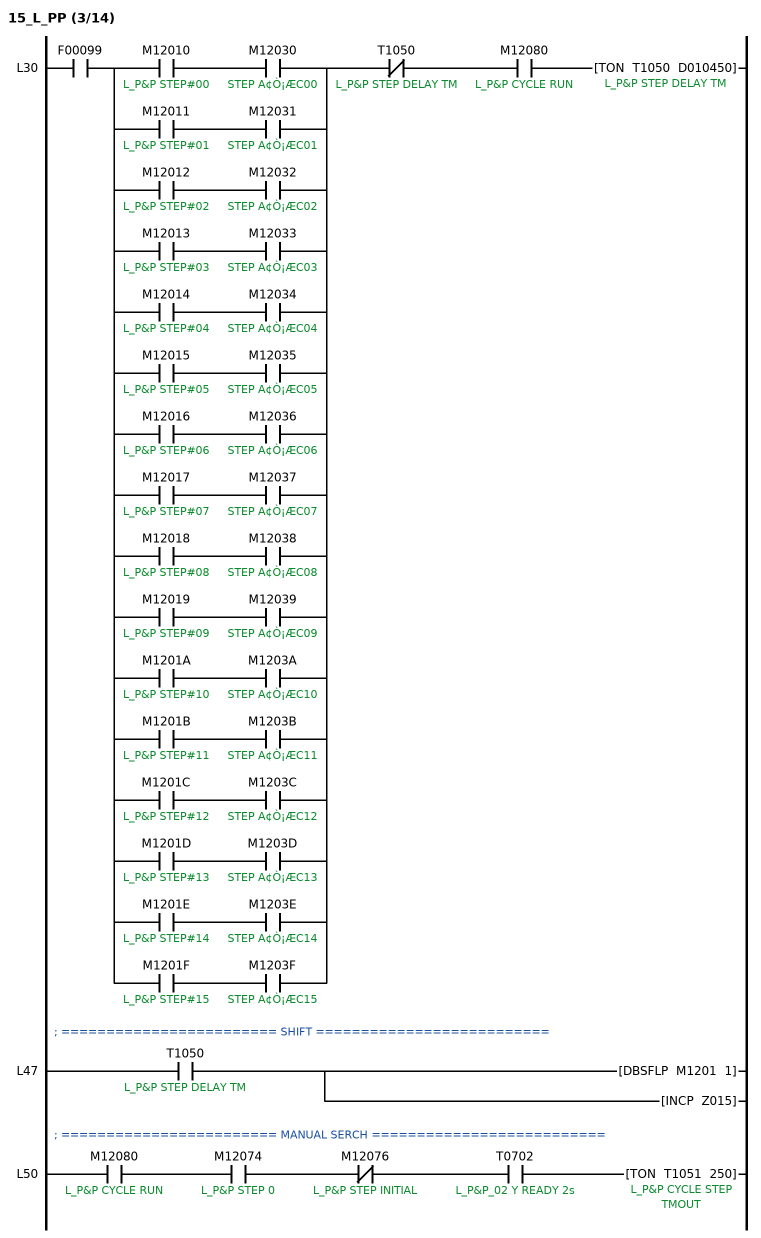
[picture p120: 15_L_PP rungs L30-L50]
; L30
LOAD      F00099
LOAD      M12010	// L_P&P STEP#00
AND       M12030	// STEP A¢Ò¡ÆC00
LOAD      M12011	// L_P&P STEP#01
AND       M12031	// STEP A¢Ò¡ÆC01
OR LOAD
LOAD      M12012	// L_P&P STEP#02
AND       M12032	// STEP A¢Ò¡ÆC02
OR LOAD
LOAD      M12013	// L_P&P STEP#03
AND       M12033	// STEP A¢Ò¡ÆC03
OR LOAD
LOAD      M12014	// L_P&P STEP#04
AND       M12034	// STEP A¢Ò¡ÆC04
OR LOAD
LOAD      M12015	// L_P&P STEP#05
AND       M12035	// STEP A¢Ò¡ÆC05
OR LOAD
LOAD      M12016	// L_P&P STEP#06
AND       M12036	// STEP A¢Ò¡ÆC06
OR LOAD
LOAD      M12017	// L_P&P STEP#07
AND       M12037	// STEP A¢Ò¡ÆC07
OR LOAD
LOAD      M12018	// L_P&P STEP#08
AND       M12038	// STEP A¢Ò¡ÆC08
OR LOAD
LOAD      M12019	// L_P&P STEP#09
AND       M12039	// STEP A¢Ò¡ÆC09
OR LOAD
LOAD      M1201A	// L_P&P STEP#10
AND       M1203A	// STEP A¢Ò¡ÆC10
OR LOAD
LOAD      M1201B	// L_P&P STEP#11
AND       M1203B	// STEP A¢Ò¡ÆC11
OR LOAD
LOAD      M1201C	// L_P&P STEP#12
AND       M1203C	// STEP A¢Ò¡ÆC12
OR LOAD
LOAD      M1201D	// L_P&P STEP#13
AND       M1203D	// STEP A¢Ò¡ÆC13
OR LOAD
LOAD      M1201E	// L_P&P STEP#14
AND       M1203E	// STEP A¢Ò¡ÆC14
OR LOAD
LOAD      M1201F	// L_P&P STEP#15
AND       M1203F	// STEP A¢Ò¡ÆC15
OR LOAD
AND LOAD
AND NOT   T1050	// L_P&P STEP DELAY TM
AND       M12080	// L_P&P CYCLE RUN
TON       T1050 D010450	// L_P&P STEP DELAY TM
// ======================== SHIFT ==========================
; L47
LOAD      T1050	// L_P&P STEP DELAY TM
DBSFLP    M1201 1
INCP      Z015
// ======================== MANUAL SERCH ==========================
; L50
LOAD      M12080	// L_P&P CYCLE RUN
AND       M12074	// L_P&P STEP 0
AND NOT   M12076	// L_P&P STEP INITIAL
AND       T0702	// L_P&P_02 Y READY 2s
TON       T1051 250	// L_P&P CYCLE STEP TMOUT

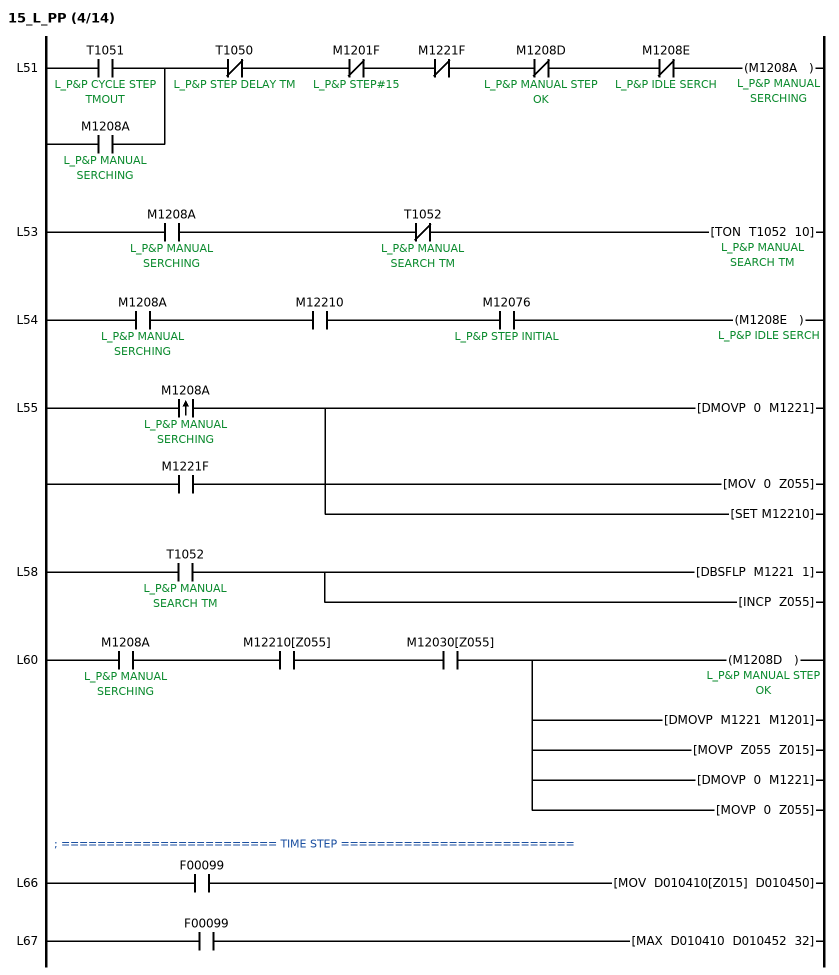
; L51
LOAD      T1051	// L_P&P CYCLE STEP TMOUT
OR        M1208A	// L_P&P MANUAL SERCHING
AND NOT   T1050	// L_P&P STEP DELAY TM
AND NOT   M1201F	// L_P&P STEP#15
AND NOT   M1221F
AND NOT   M1208D	// L_P&P MANUAL STEP OK
AND NOT   M1208E	// L_P&P IDLE SERCH
OUT       M1208A	// L_P&P MANUAL SERCHING
; L53
LOAD      M1208A	// L_P&P MANUAL SERCHING
AND NOT   T1052	// L_P&P MANUAL SEARCH TM
TON       T1052 10	// L_P&P MANUAL SEARCH TM
; L54
LOAD      M1208A	// L_P&P MANUAL SERCHING
AND       M12210
AND       M12076	// L_P&P STEP INITIAL
OUT       M1208E	// L_P&P IDLE SERCH
; L55
LOADP     M1208A	// L_P&P MANUAL SERCHING
OR        M1221F
DMOVP     0 M1221
MOV       0 Z055
SET       M12210
; L58
LOAD      T1052	// L_P&P MANUAL SEARCH TM
DBSFLP    M1221 1
INCP      Z055
; L60
LOAD      M1208A	// L_P&P MANUAL SERCHING
AND       M12210[Z055]
AND       M12030[Z055]
OUT       M1208D	// L_P&P MANUAL STEP OK
DMOVP     M1221 M1201
MOVP      Z055 Z015
DMOVP     0 M1221
MOVP      0 Z055
// ======================== TIME STEP ==========================
; L66
LOAD      F00099
MOV       D010410[Z015] D010450
; L67
LOAD      F00099
MAX       D010410 D010452 32

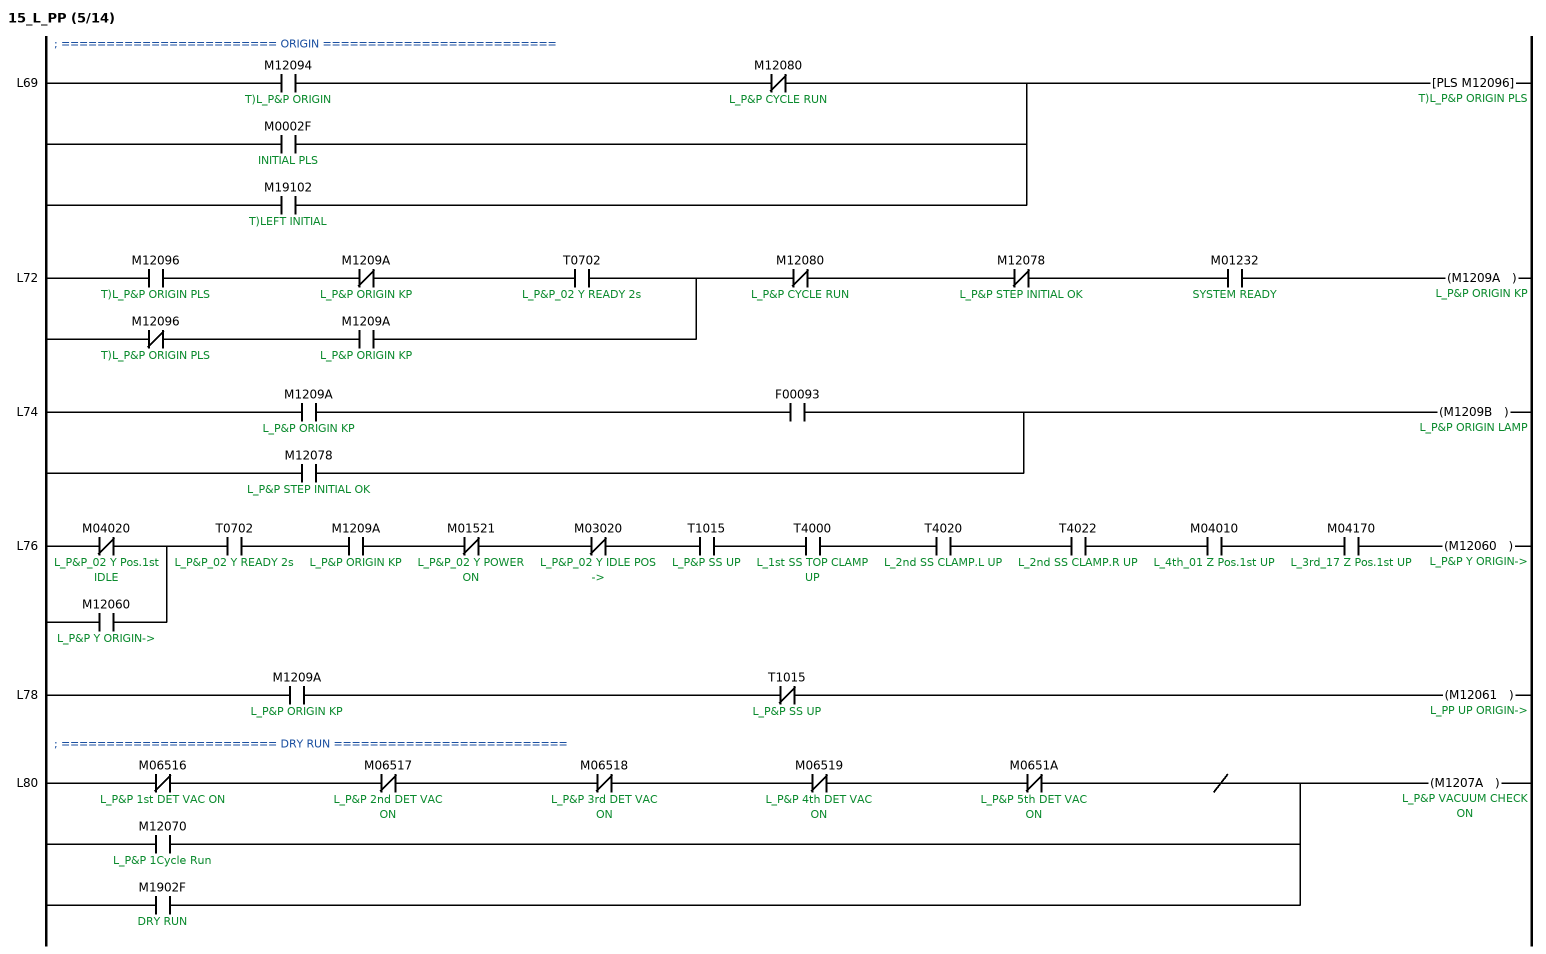
// ======================== ORIGIN ==========================
; L69
LOAD      M12094	// T)L_P&P ORIGIN
AND NOT   M12080	// L_P&P CYCLE RUN
OR        M0002F	// INITIAL PLS
OR        M19102	// T)LEFT INITIAL
OUTP      M12096	// T)L_P&P ORIGIN PLS
; L72
LOAD      M12096	// T)L_P&P ORIGIN PLS
AND NOT   M1209A	// L_P&P ORIGIN KP
AND       T0702	// L_P&P_02 Y READY 2s
LOAD NOT  M12096	// T)L_P&P ORIGIN PLS
AND       M1209A	// L_P&P ORIGIN KP
OR LOAD
AND NOT   M12080	// L_P&P CYCLE RUN
AND NOT   M12078	// L_P&P STEP INITIAL OK
AND       M01232	// SYSTEM READY
OUT       M1209A	// L_P&P ORIGIN KP
; L74
LOAD      M1209A	// L_P&P ORIGIN KP
AND       F00093
OR        M12078	// L_P&P STEP INITIAL OK
OUT       M1209B	// L_P&P ORIGIN LAMP
; L76
LOAD NOT  M04020	// L_P&P_02 Y Pos.1st IDLE
OR        M12060	// L_P&P Y ORIGIN->
AND       T0702	// L_P&P_02 Y READY 2s
AND       M1209A	// L_P&P ORIGIN KP
AND NOT   M01521	// L_P&P_02 Y POWER ON
AND NOT   M03020	// L_P&P_02 Y IDLE POS ->
AND       T1015	// L_P&P SS UP
AND       T4000	// L_1st SS TOP CLAMP    UP
AND       T4020	// L_2nd SS CLAMP.L UP
AND       T4022	// L_2nd SS CLAMP.R UP
AND       M04010	// L_4th_01 Z Pos.1st UP
AND       M04170	// L_3rd_17 Z Pos.1st UP
OUT       M12060	// L_P&P Y ORIGIN->
; L78
LOAD      M1209A	// L_P&P ORIGIN KP
AND NOT   T1015	// L_P&P SS UP
OUT       M12061	// L_PP UP ORIGIN->
// ======================== DRY RUN ==========================
; L80
LOAD NOT  M06516	// L_P&P 1st DET VAC ON
AND NOT   M06517	// L_P&P 2nd DET VAC ON
AND NOT   M06518	// L_P&P 3rd DET VAC ON
AND NOT   M06519	// L_P&P 4th DET VAC ON
AND NOT   M0651A	// L_P&P 5th DET VAC ON
NOT
OR        M12070	// L_P&P 1Cycle Run
OR        M1902F	// DRY RUN
OUT       M1207A	// L_P&P VACUUM CHECK ON

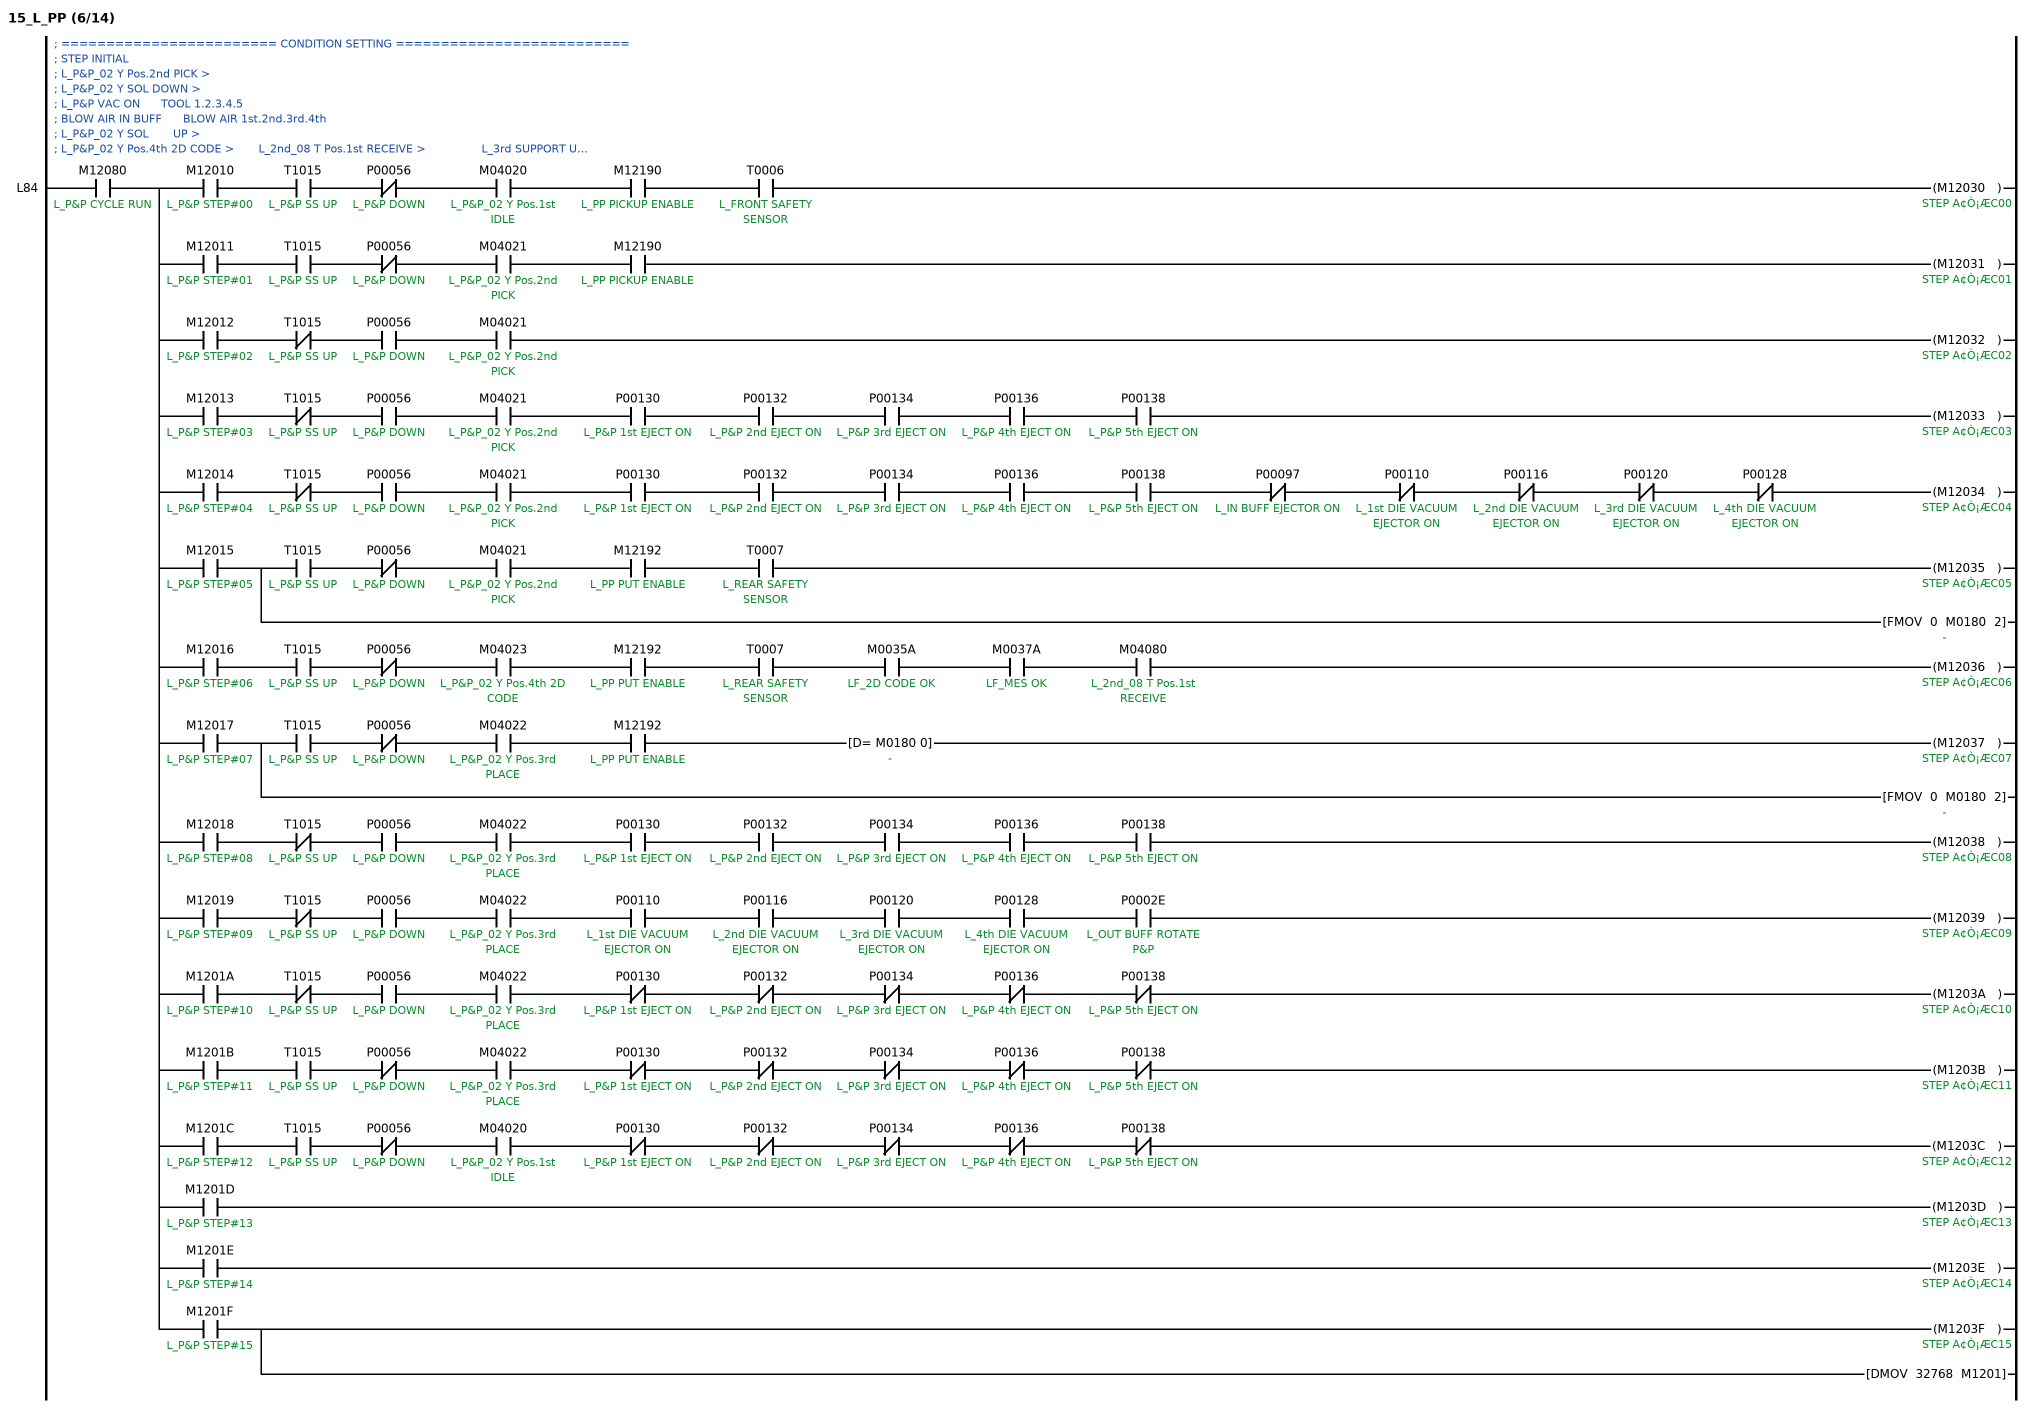
// ======================== CONDITION SETTING ==========================
; L84
LOAD      M12080	// L_P&P CYCLE RUN
MPUSH
AND       M12010	// L_P&P STEP#00
AND       T1015	// L_P&P SS UP
AND NOT   P00056	// L_P&P DOWN
AND       M04020	// L_P&P_02 Y Pos.1st IDLE
AND       M12190	// L_PP PICKUP ENABLE
AND       T0006	// L_FRONT SAFETY SENSOR
OUT       M12030	// STEP A¢Ò¡ÆC00
MLOAD
AND       M12011	// L_P&P STEP#01
AND       T1015	// L_P&P SS UP
AND NOT   P00056	// L_P&P DOWN
AND       M04021	// L_P&P_02 Y Pos.2nd PICK
AND       M12190	// L_PP PICKUP ENABLE
OUT       M12031	// STEP A¢Ò¡ÆC01
MLOAD
AND       M12012	// L_P&P STEP#02
AND NOT   T1015	// L_P&P SS UP
AND       P00056	// L_P&P DOWN
AND       M04021	// L_P&P_02 Y Pos.2nd PICK
OUT       M12032	// STEP A¢Ò¡ÆC02
MLOAD
AND       M12013	// L_P&P STEP#03
AND NOT   T1015	// L_P&P SS UP
AND       P00056	// L_P&P DOWN
AND       M04021	// L_P&P_02 Y Pos.2nd PICK
AND       P00130	// L_P&P 1st EJECT ON
AND       P00132	// L_P&P 2nd EJECT ON
AND       P00134	// L_P&P 3rd EJECT ON
AND       P00136	// L_P&P 4th EJECT ON
AND       P00138	// L_P&P 5th EJECT ON
OUT       M12033	// STEP A¢Ò¡ÆC03
MLOAD
AND       M12014	// L_P&P STEP#04
AND NOT   T1015	// L_P&P SS UP
AND       P00056	// L_P&P DOWN
AND       M04021	// L_P&P_02 Y Pos.2nd PICK
AND       P00130	// L_P&P 1st EJECT ON
AND       P00132	// L_P&P 2nd EJECT ON
AND       P00134	// L_P&P 3rd EJECT ON
AND       P00136	// L_P&P 4th EJECT ON
AND       P00138	// L_P&P 5th EJECT ON
AND NOT   P00097	// L_IN BUFF EJECTOR ON
AND NOT   P00110	// L_1st DIE VACUUM EJECTOR ON
AND NOT   P00116	// L_2nd DIE VACUUM EJECTOR ON
AND NOT   P00120	// L_3rd DIE VACUUM EJECTOR ON
AND NOT   P00128	// L_4th DIE VACUUM EJECTOR ON
OUT       M12034	// STEP A¢Ò¡ÆC04
MLOAD
AND       M12015	// L_P&P STEP#05
MPUSH
AND       T1015	// L_P&P SS UP
AND NOT   P00056	// L_P&P DOWN
AND       M04021	// L_P&P_02 Y Pos.2nd PICK
AND       M12192	// L_PP PUT ENABLE
AND       T0007	// L_REAR SAFETY SENSOR
OUT       M12035	// STEP A¢Ò¡ÆC05
MPOP
FMOV      0 M0180 2	// -
MLOAD
AND       M12016	// L_P&P STEP#06
AND       T1015	// L_P&P SS UP
AND NOT   P00056	// L_P&P DOWN
AND       M04023	// L_P&P_02 Y Pos.4th 2D CODE
AND       M12192	// L_PP PUT ENABLE
AND       T0007	// L_REAR SAFETY SENSOR
AND       M0035A	// LF_2D CODE OK
AND       M0037A	// LF_MES OK
AND       M04080	// L_2nd_08 T Pos.1st RECEIVE
OUT       M12036	// STEP A¢Ò¡ÆC06
MLOAD
AND       M12017	// L_P&P STEP#07
MPUSH
AND       T1015	// L_P&P SS UP
AND NOT   P00056	// L_P&P DOWN
AND       M04022	// L_P&P_02 Y Pos.3rd PLACE
AND       M12192	// L_PP PUT ENABLE
ANDD=     M0180 0	// -
OUT       M12037	// STEP A¢Ò¡ÆC07
MPOP
FMOV      0 M0180 2	// -
MLOAD
AND       M12018	// L_P&P STEP#08
AND NOT   T1015	// L_P&P SS UP
AND       P00056	// L_P&P DOWN
AND       M04022	// L_P&P_02 Y Pos.3rd PLACE
AND       P00130	// L_P&P 1st EJECT ON
AND       P00132	// L_P&P 2nd EJECT ON
AND       P00134	// L_P&P 3rd EJECT ON
AND       P00136	// L_P&P 4th EJECT ON
AND       P00138	// L_P&P 5th EJECT ON
OUT       M12038	// STEP A¢Ò¡ÆC08
MLOAD
AND       M12019	// L_P&P STEP#09
AND NOT   T1015	// L_P&P SS UP
AND       P00056	// L_P&P DOWN
AND       M04022	// L_P&P_02 Y Pos.3rd PLACE
AND       P00110	// L_1st DIE VACUUM EJECTOR ON
AND       P00116	// L_2nd DIE VACUUM EJECTOR ON
AND       P00120	// L_3rd DIE VACUUM EJECTOR ON
AND       P00128	// L_4th DIE VACUUM EJECTOR ON
AND       P0002E	// L_OUT BUFF ROTATE      P&P
OUT       M12039	// STEP A¢Ò¡ÆC09
MLOAD
AND       M1201A	// L_P&P STEP#10
AND NOT   T1015	// L_P&P SS UP
AND       P00056	// L_P&P DOWN
AND       M04022	// L_P&P_02 Y Pos.3rd PLACE
AND NOT   P00130	// L_P&P 1st EJECT ON
AND NOT   P00132	// L_P&P 2nd EJECT ON
AND NOT   P00134	// L_P&P 3rd EJECT ON
AND NOT   P00136	// L_P&P 4th EJECT ON
AND NOT   P00138	// L_P&P 5th EJECT ON
OUT       M1203A	// STEP A¢Ò¡ÆC10
MLOAD
AND       M1201B	// L_P&P STEP#11
AND       T1015	// L_P&P SS UP
AND NOT   P00056	// L_P&P DOWN
AND       M04022	// L_P&P_02 Y Pos.3rd PLACE
AND NOT   P00130	// L_P&P 1st EJECT ON
AND NOT   P00132	// L_P&P 2nd EJECT ON
AND NOT   P00134	// L_P&P 3rd EJECT ON
AND NOT   P00136	// L_P&P 4th EJECT ON
AND NOT   P00138	// L_P&P 5th EJECT ON
OUT       M1203B	// STEP A¢Ò¡ÆC11
MLOAD
AND       M1201C	// L_P&P STEP#12
AND       T1015	// L_P&P SS UP
AND NOT   P00056	// L_P&P DOWN
AND       M04020	// L_P&P_02 Y Pos.1st IDLE
AND NOT   P00130	// L_P&P 1st EJECT ON
AND NOT   P00132	// L_P&P 2nd EJECT ON
AND NOT   P00134	// L_P&P 3rd EJECT ON
AND NOT   P00136	// L_P&P 4th EJECT ON
AND NOT   P00138	// L_P&P 5th EJECT ON
OUT       M1203C	// STEP A¢Ò¡ÆC12
MLOAD
AND       M1201D	// L_P&P STEP#13
OUT       M1203D	// STEP A¢Ò¡ÆC13
MLOAD
AND       M1201E	// L_P&P STEP#14
OUT       M1203E	// STEP A¢Ò¡ÆC14
MPOP
AND       M1201F	// L_P&P STEP#15
OUT       M1203F	// STEP A¢Ò¡ÆC15
DMOV      32768 M1201
// output comment: STEP INITIAL
// output comment: L_P&P_02 Y Pos.2nd PICK >
// output comment: L_P&P_02 Y SOL DOWN >
// output comment: L_P&P VAC ON      TOOL 1.2.3.4.5
// output comment: BLOW AIR IN BUFF      BLOW AIR 1st.2nd.3rd.4th
// output comment: L_P&P_02 Y SOL       UP >
// output comment: L_P&P_02 Y Pos.4th 2D CODE >       L_2nd_08 T Pos.1st RECEIVE >                L_3rd SUPPORT UP
// output comment: L_P&P_02 Y Pos.3rd PLACE >
// output comment: L_P&P_02 Y SOL       DOWN >
// output comment: L_P&P BLOW AIR      TOOL 1.2.3.4.5
// output comment: L_P&P_02 Y SOL       UP >
// output comment: L_P&P_02 Y Pos.1st IDLE >

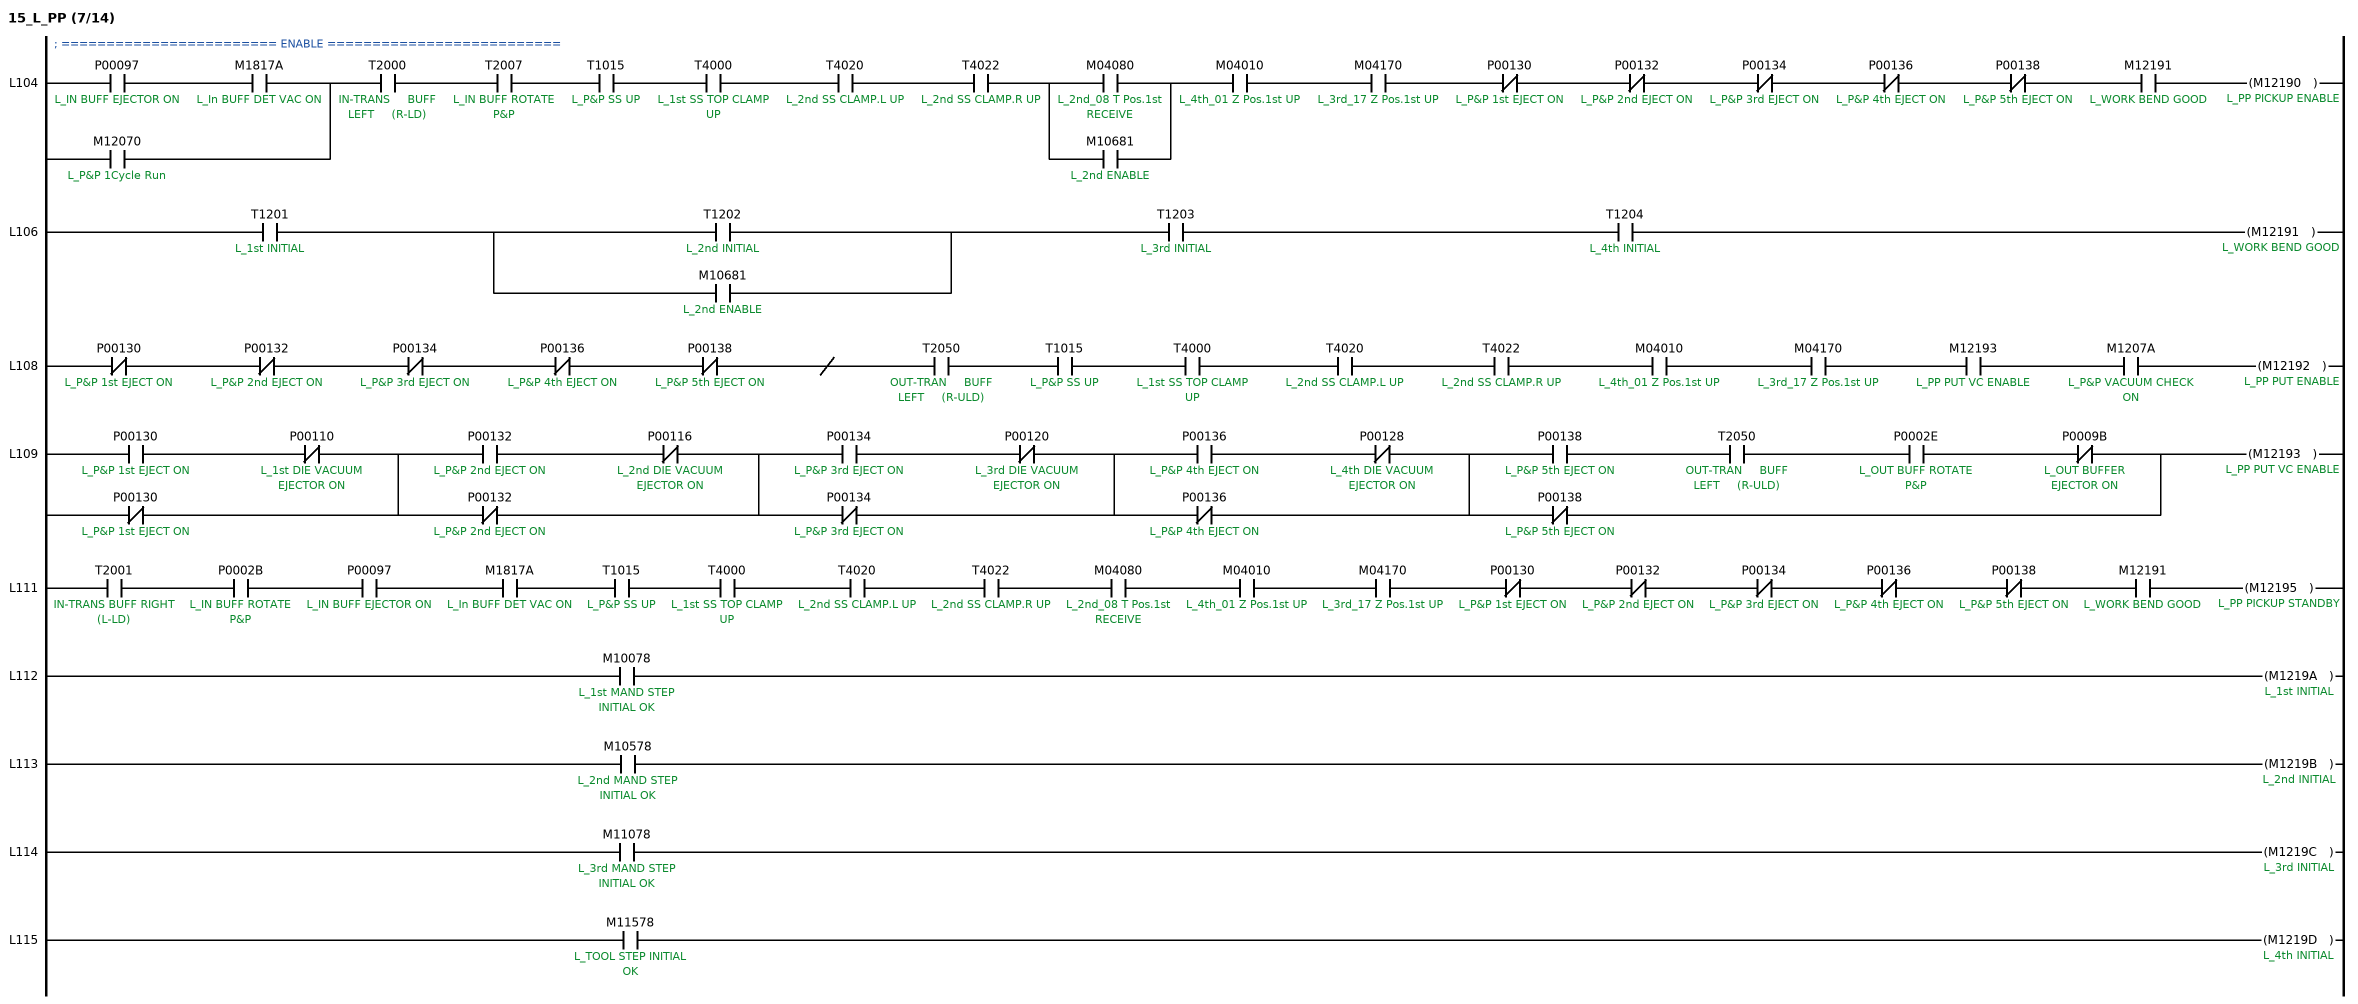
// ======================== ENABLE ==========================
; L104
LOAD      P00097	// L_IN BUFF EJECTOR ON
AND       M1817A	// L_In BUFF DET VAC ON
OR        M12070	// L_P&P 1Cycle Run
AND       T2000	// IN-TRANS     BUFF     LEFT     (R-LD)
AND       T2007	// L_IN BUFF ROTATE      P&P
AND       T1015	// L_P&P SS UP
AND       T4000	// L_1st SS TOP CLAMP    UP
AND       T4020	// L_2nd SS CLAMP.L UP
AND       T4022	// L_2nd SS CLAMP.R UP
LOAD      M04080	// L_2nd_08 T Pos.1st RECEIVE
OR        M10681	// L_2nd ENABLE
AND LOAD
AND       M04010	// L_4th_01 Z Pos.1st UP
AND       M04170	// L_3rd_17 Z Pos.1st UP
AND NOT   P00130	// L_P&P 1st EJECT ON
AND NOT   P00132	// L_P&P 2nd EJECT ON
AND NOT   P00134	// L_P&P 3rd EJECT ON
AND NOT   P00136	// L_P&P 4th EJECT ON
AND NOT   P00138	// L_P&P 5th EJECT ON
AND       M12191	// L_WORK BEND GOOD
OUT       M12190	// L_PP PICKUP ENABLE
; L106
LOAD      T1201	// L_1st INITIAL
LOAD      T1202	// L_2nd INITIAL
OR        M10681	// L_2nd ENABLE
AND LOAD
AND       T1203	// L_3rd INITIAL
AND       T1204	// L_4th INITIAL
OUT       M12191	// L_WORK BEND GOOD
; L108
LOAD NOT  P00130	// L_P&P 1st EJECT ON
AND NOT   P00132	// L_P&P 2nd EJECT ON
AND NOT   P00134	// L_P&P 3rd EJECT ON
AND NOT   P00136	// L_P&P 4th EJECT ON
AND NOT   P00138	// L_P&P 5th EJECT ON
NOT
AND       T2050	// OUT-TRAN     BUFF     LEFT     (R-ULD)
AND       T1015	// L_P&P SS UP
AND       T4000	// L_1st SS TOP CLAMP    UP
AND       T4020	// L_2nd SS CLAMP.L UP
AND       T4022	// L_2nd SS CLAMP.R UP
AND       M04010	// L_4th_01 Z Pos.1st UP
AND       M04170	// L_3rd_17 Z Pos.1st UP
AND       M12193	// L_PP PUT VC ENABLE
AND       M1207A	// L_P&P VACUUM CHECK ON
OUT       M12192	// L_PP PUT ENABLE
; L109
LOAD      P00130	// L_P&P 1st EJECT ON
AND NOT   P00110	// L_1st DIE VACUUM EJECTOR ON
OR NOT    P00130	// L_P&P 1st EJECT ON
LOAD      P00132	// L_P&P 2nd EJECT ON
AND NOT   P00116	// L_2nd DIE VACUUM EJECTOR ON
OR NOT    P00132	// L_P&P 2nd EJECT ON
AND LOAD
LOAD      P00134	// L_P&P 3rd EJECT ON
AND NOT   P00120	// L_3rd DIE VACUUM EJECTOR ON
OR NOT    P00134	// L_P&P 3rd EJECT ON
AND LOAD
LOAD      P00136	// L_P&P 4th EJECT ON
AND NOT   P00128	// L_4th DIE VACUUM EJECTOR ON
OR NOT    P00136	// L_P&P 4th EJECT ON
AND LOAD
LOAD      P00138	// L_P&P 5th EJECT ON
AND       T2050	// OUT-TRAN     BUFF     LEFT     (R-ULD)
AND       P0002E	// L_OUT BUFF ROTATE      P&P
AND NOT   P0009B	// L_OUT BUFFER EJECTOR ON
OR NOT    P00138	// L_P&P 5th EJECT ON
AND LOAD
OUT       M12193	// L_PP PUT VC ENABLE
; L111
LOAD      T2001	// IN-TRANS BUFF RIGHT     (L-LD)
AND       P0002B	// L_IN BUFF ROTATE      P&P
AND       P00097	// L_IN BUFF EJECTOR ON
AND       M1817A	// L_In BUFF DET VAC ON
AND       T1015	// L_P&P SS UP
AND       T4000	// L_1st SS TOP CLAMP    UP
AND       T4020	// L_2nd SS CLAMP.L UP
AND       T4022	// L_2nd SS CLAMP.R UP
AND       M04080	// L_2nd_08 T Pos.1st RECEIVE
AND       M04010	// L_4th_01 Z Pos.1st UP
AND       M04170	// L_3rd_17 Z Pos.1st UP
AND NOT   P00130	// L_P&P 1st EJECT ON
AND NOT   P00132	// L_P&P 2nd EJECT ON
AND NOT   P00134	// L_P&P 3rd EJECT ON
AND NOT   P00136	// L_P&P 4th EJECT ON
AND NOT   P00138	// L_P&P 5th EJECT ON
AND       M12191	// L_WORK BEND GOOD
OUT       M12195	// L_PP PICKUP STANDBY
; L112
LOAD      M10078	// L_1st MAND STEP INITIAL OK
OUT       M1219A	// L_1st INITIAL
; L113
LOAD      M10578	// L_2nd MAND STEP INITIAL OK
OUT       M1219B	// L_2nd INITIAL
; L114
LOAD      M11078	// L_3rd MAND STEP INITIAL OK
OUT       M1219C	// L_3rd INITIAL
; L115
LOAD      M11578	// L_TOOL STEP INITIAL OK
OUT       M1219D	// L_4th INITIAL

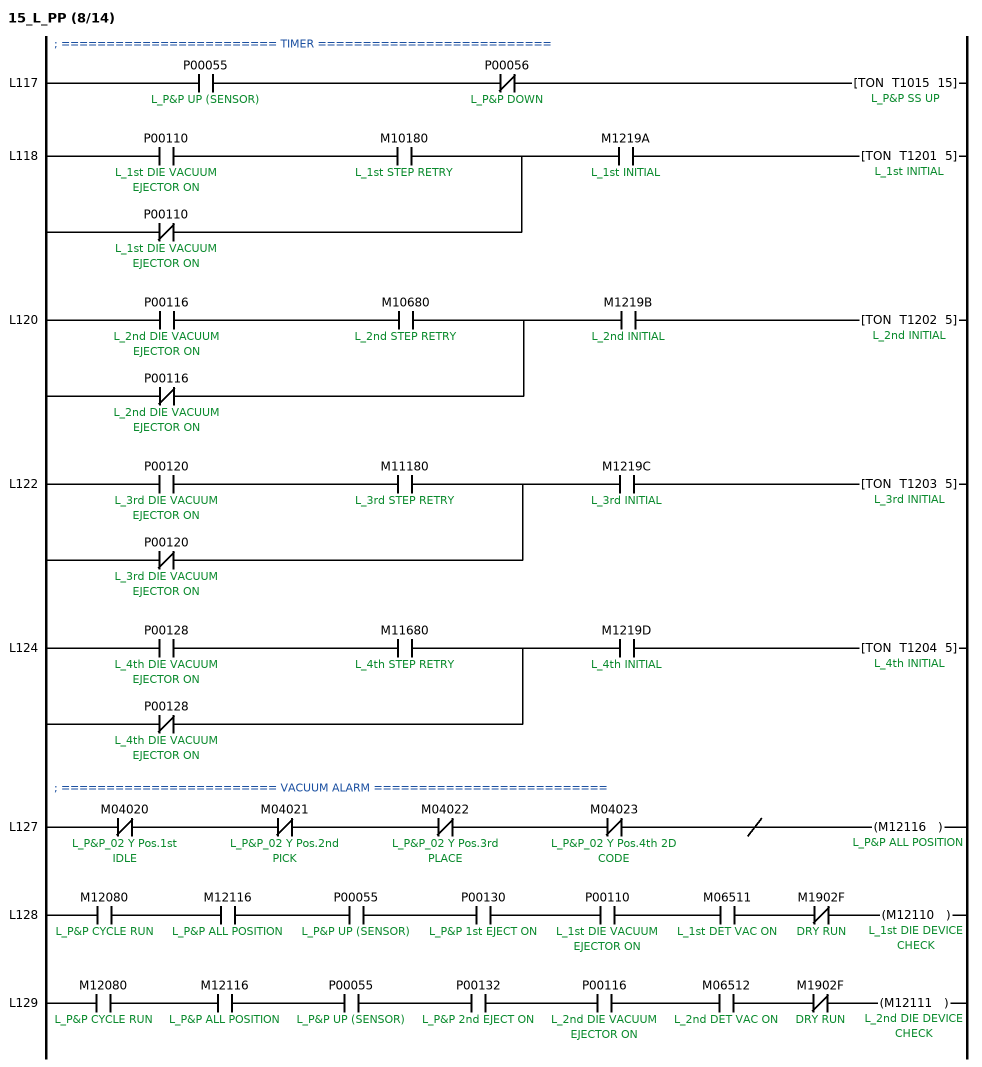
// ======================== TIMER ==========================
; L117
LOAD      P00055	// L_P&P UP (SENSOR)
AND NOT   P00056	// L_P&P DOWN
TON       T1015 15	// L_P&P SS UP
; L118
LOAD      P00110	// L_1st DIE VACUUM EJECTOR ON
AND       M10180	// L_1st STEP RETRY
OR NOT    P00110	// L_1st DIE VACUUM EJECTOR ON
AND       M1219A	// L_1st INITIAL
TON       T1201 5	// L_1st INITIAL
; L120
LOAD      P00116	// L_2nd DIE VACUUM EJECTOR ON
AND       M10680	// L_2nd STEP RETRY
OR NOT    P00116	// L_2nd DIE VACUUM EJECTOR ON
AND       M1219B	// L_2nd INITIAL
TON       T1202 5	// L_2nd INITIAL
; L122
LOAD      P00120	// L_3rd DIE VACUUM EJECTOR ON
AND       M11180	// L_3rd STEP RETRY
OR NOT    P00120	// L_3rd DIE VACUUM EJECTOR ON
AND       M1219C	// L_3rd INITIAL
TON       T1203 5	// L_3rd INITIAL
; L124
LOAD      P00128	// L_4th DIE VACUUM EJECTOR ON
AND       M11680	// L_4th STEP RETRY
OR NOT    P00128	// L_4th DIE VACUUM EJECTOR ON
AND       M1219D	// L_4th INITIAL
TON       T1204 5	// L_4th INITIAL
// ======================== VACUUM ALARM ==========================
; L127
LOAD NOT  M04020	// L_P&P_02 Y Pos.1st IDLE
AND NOT   M04021	// L_P&P_02 Y Pos.2nd PICK
AND NOT   M04022	// L_P&P_02 Y Pos.3rd PLACE
AND NOT   M04023	// L_P&P_02 Y Pos.4th 2D CODE
NOT
OUT       M12116	// L_P&P ALL POSITION
; L128
LOAD      M12080	// L_P&P CYCLE RUN
AND       M12116	// L_P&P ALL POSITION
AND       P00055	// L_P&P UP (SENSOR)
AND       P00130	// L_P&P 1st EJECT ON
AND       P00110	// L_1st DIE VACUUM EJECTOR ON
AND       M06511	// L_1st DET VAC ON
AND NOT   M1902F	// DRY RUN
OUT       M12110	// L_1st DIE DEVICE CHECK
; L129
LOAD      M12080	// L_P&P CYCLE RUN
AND       M12116	// L_P&P ALL POSITION
AND       P00055	// L_P&P UP (SENSOR)
AND       P00132	// L_P&P 2nd EJECT ON
AND       P00116	// L_2nd DIE VACUUM EJECTOR ON
AND       M06512	// L_2nd DET VAC ON
AND NOT   M1902F	// DRY RUN
OUT       M12111	// L_2nd DIE DEVICE CHECK

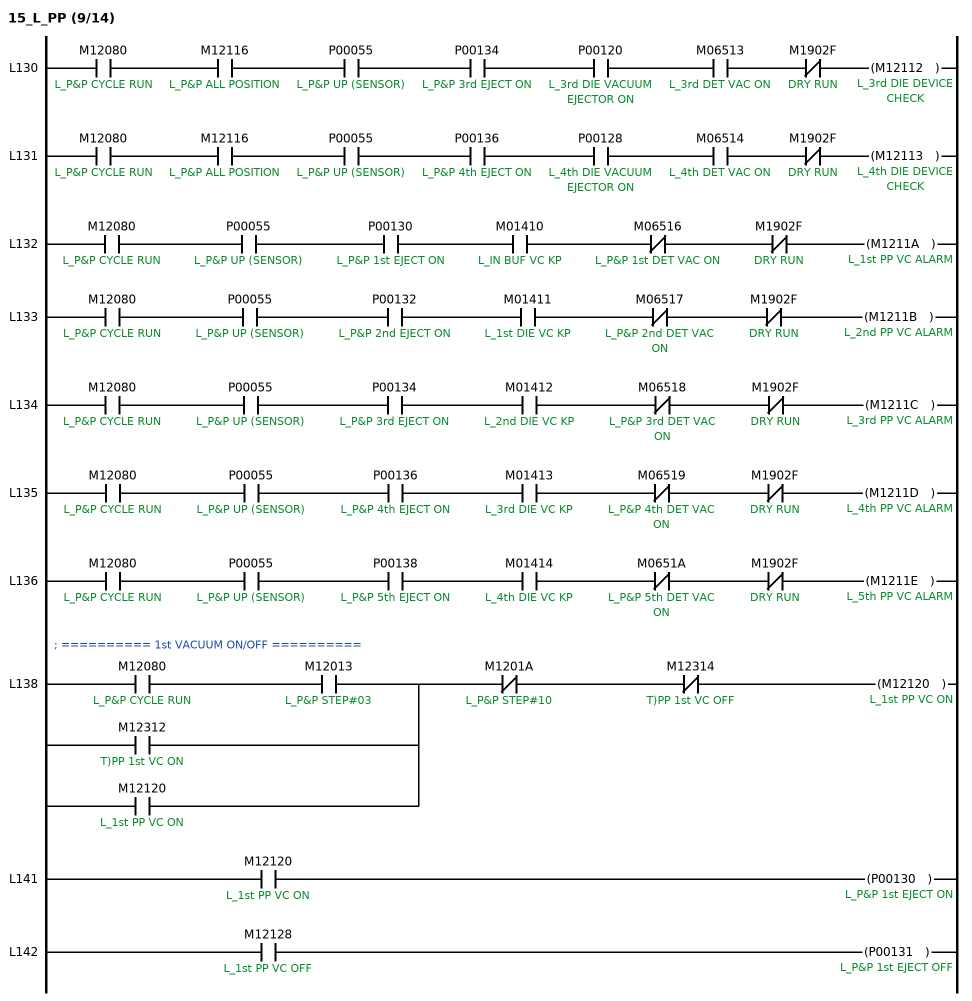
; L130
LOAD      M12080	// L_P&P CYCLE RUN
AND       M12116	// L_P&P ALL POSITION
AND       P00055	// L_P&P UP (SENSOR)
AND       P00134	// L_P&P 3rd EJECT ON
AND       P00120	// L_3rd DIE VACUUM EJECTOR ON
AND       M06513	// L_3rd DET VAC ON
AND NOT   M1902F	// DRY RUN
OUT       M12112	// L_3rd DIE DEVICE CHECK
; L131
LOAD      M12080	// L_P&P CYCLE RUN
AND       M12116	// L_P&P ALL POSITION
AND       P00055	// L_P&P UP (SENSOR)
AND       P00136	// L_P&P 4th EJECT ON
AND       P00128	// L_4th DIE VACUUM EJECTOR ON
AND       M06514	// L_4th DET VAC ON
AND NOT   M1902F	// DRY RUN
OUT       M12113	// L_4th DIE DEVICE CHECK
; L132
LOAD      M12080	// L_P&P CYCLE RUN
AND       P00055	// L_P&P UP (SENSOR)
AND       P00130	// L_P&P 1st EJECT ON
AND       M01410	// L_IN BUF VC KP
AND NOT   M06516	// L_P&P 1st DET VAC ON
AND NOT   M1902F	// DRY RUN
OUT       M1211A	// L_1st PP VC ALARM
; L133
LOAD      M12080	// L_P&P CYCLE RUN
AND       P00055	// L_P&P UP (SENSOR)
AND       P00132	// L_P&P 2nd EJECT ON
AND       M01411	// L_1st DIE VC KP
AND NOT   M06517	// L_P&P 2nd DET VAC ON
AND NOT   M1902F	// DRY RUN
OUT       M1211B	// L_2nd PP VC ALARM
; L134
LOAD      M12080	// L_P&P CYCLE RUN
AND       P00055	// L_P&P UP (SENSOR)
AND       P00134	// L_P&P 3rd EJECT ON
AND       M01412	// L_2nd DIE VC KP
AND NOT   M06518	// L_P&P 3rd DET VAC ON
AND NOT   M1902F	// DRY RUN
OUT       M1211C	// L_3rd PP VC ALARM
; L135
LOAD      M12080	// L_P&P CYCLE RUN
AND       P00055	// L_P&P UP (SENSOR)
AND       P00136	// L_P&P 4th EJECT ON
AND       M01413	// L_3rd DIE VC KP
AND NOT   M06519	// L_P&P 4th DET VAC ON
AND NOT   M1902F	// DRY RUN
OUT       M1211D	// L_4th PP VC ALARM
; L136
LOAD      M12080	// L_P&P CYCLE RUN
AND       P00055	// L_P&P UP (SENSOR)
AND       P00138	// L_P&P 5th EJECT ON
AND       M01414	// L_4th DIE VC KP
AND NOT   M0651A	// L_P&P 5th DET VAC ON
AND NOT   M1902F	// DRY RUN
OUT       M1211E	// L_5th PP VC ALARM
// ========== 1st VACUUM ON/OFF ==========
; L138
LOAD      M12080	// L_P&P CYCLE RUN
AND       M12013	// L_P&P STEP#03
OR        M12312	// T)PP 1st VC ON
OR        M12120	// L_1st PP VC ON
AND NOT   M1201A	// L_P&P STEP#10
AND NOT   M12314	// T)PP 1st VC OFF
OUT       M12120	// L_1st PP VC ON
; L141
LOAD      M12120	// L_1st PP VC ON
OUT       P00130	// L_P&P 1st EJECT ON
; L142
LOAD      M12128	// L_1st PP VC OFF
OUT       P00131	// L_P&P 1st EJECT OFF

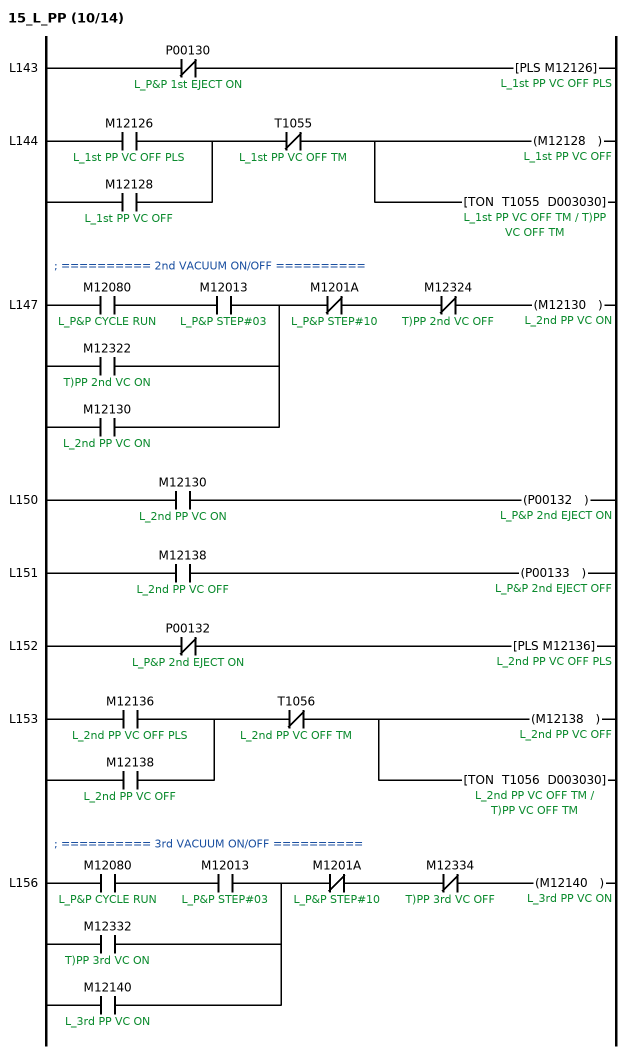
; L143
LOAD NOT  P00130	// L_P&P 1st EJECT ON
OUTP      M12126	// L_1st PP VC OFF PLS
; L144
LOAD      M12126	// L_1st PP VC OFF PLS
OR        M12128	// L_1st PP VC OFF
AND NOT   T1055	// L_1st PP VC OFF TM
OUT       M12128	// L_1st PP VC OFF
TON       T1055 D003030	// L_1st PP VC OFF TM / T)PP VC OFF TM
// ========== 2nd VACUUM ON/OFF ==========
; L147
LOAD      M12080	// L_P&P CYCLE RUN
AND       M12013	// L_P&P STEP#03
OR        M12322	// T)PP 2nd VC ON
OR        M12130	// L_2nd PP VC ON
AND NOT   M1201A	// L_P&P STEP#10
AND NOT   M12324	// T)PP 2nd VC OFF
OUT       M12130	// L_2nd PP VC ON
; L150
LOAD      M12130	// L_2nd PP VC ON
OUT       P00132	// L_P&P 2nd EJECT ON
; L151
LOAD      M12138	// L_2nd PP VC OFF
OUT       P00133	// L_P&P 2nd EJECT OFF
; L152
LOAD NOT  P00132	// L_P&P 2nd EJECT ON
OUTP      M12136	// L_2nd PP VC OFF PLS
; L153
LOAD      M12136	// L_2nd PP VC OFF PLS
OR        M12138	// L_2nd PP VC OFF
AND NOT   T1056	// L_2nd PP VC OFF TM
OUT       M12138	// L_2nd PP VC OFF
TON       T1056 D003030	// L_2nd PP VC OFF TM / T)PP VC OFF TM
// ========== 3rd VACUUM ON/OFF ==========
; L156
LOAD      M12080	// L_P&P CYCLE RUN
AND       M12013	// L_P&P STEP#03
OR        M12332	// T)PP 3rd VC ON
OR        M12140	// L_3rd PP VC ON
AND NOT   M1201A	// L_P&P STEP#10
AND NOT   M12334	// T)PP 3rd VC OFF
OUT       M12140	// L_3rd PP VC ON

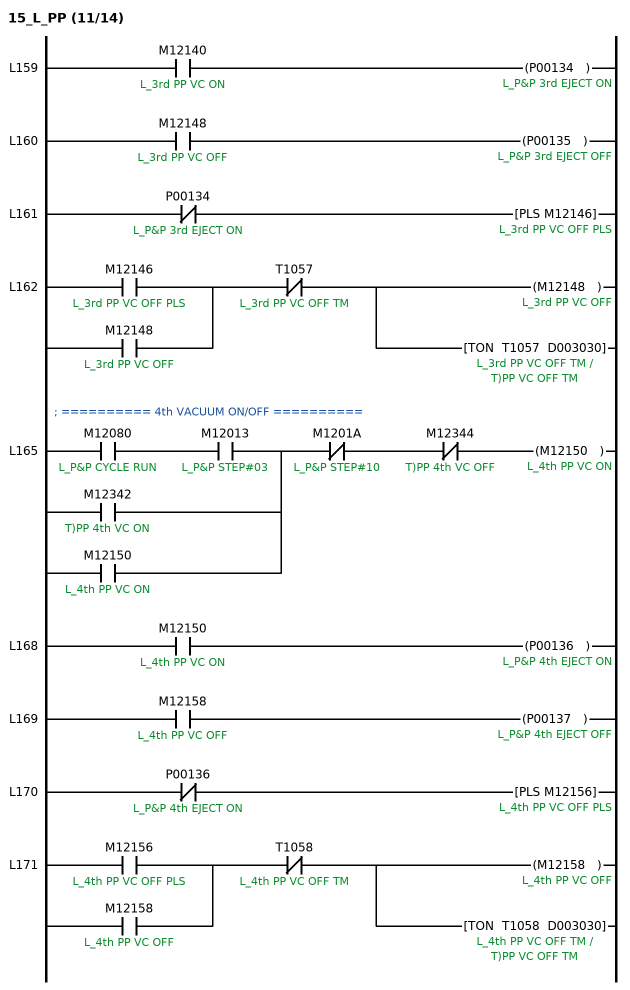
; L159
LOAD      M12140	// L_3rd PP VC ON
OUT       P00134	// L_P&P 3rd EJECT ON
; L160
LOAD      M12148	// L_3rd PP VC OFF
OUT       P00135	// L_P&P 3rd EJECT OFF
; L161
LOAD NOT  P00134	// L_P&P 3rd EJECT ON
OUTP      M12146	// L_3rd PP VC OFF PLS
; L162
LOAD      M12146	// L_3rd PP VC OFF PLS
OR        M12148	// L_3rd PP VC OFF
AND NOT   T1057	// L_3rd PP VC OFF TM
OUT       M12148	// L_3rd PP VC OFF
TON       T1057 D003030	// L_3rd PP VC OFF TM / T)PP VC OFF TM
// ========== 4th VACUUM ON/OFF ==========
; L165
LOAD      M12080	// L_P&P CYCLE RUN
AND       M12013	// L_P&P STEP#03
OR        M12342	// T)PP 4th VC ON
OR        M12150	// L_4th PP VC ON
AND NOT   M1201A	// L_P&P STEP#10
AND NOT   M12344	// T)PP 4th VC OFF
OUT       M12150	// L_4th PP VC ON
; L168
LOAD      M12150	// L_4th PP VC ON
OUT       P00136	// L_P&P 4th EJECT ON
; L169
LOAD      M12158	// L_4th PP VC OFF
OUT       P00137	// L_P&P 4th EJECT OFF
; L170
LOAD NOT  P00136	// L_P&P 4th EJECT ON
OUTP      M12156	// L_4th PP VC OFF PLS
; L171
LOAD      M12156	// L_4th PP VC OFF PLS
OR        M12158	// L_4th PP VC OFF
AND NOT   T1058	// L_4th PP VC OFF TM
OUT       M12158	// L_4th PP VC OFF
TON       T1058 D003030	// L_4th PP VC OFF TM / T)PP VC OFF TM

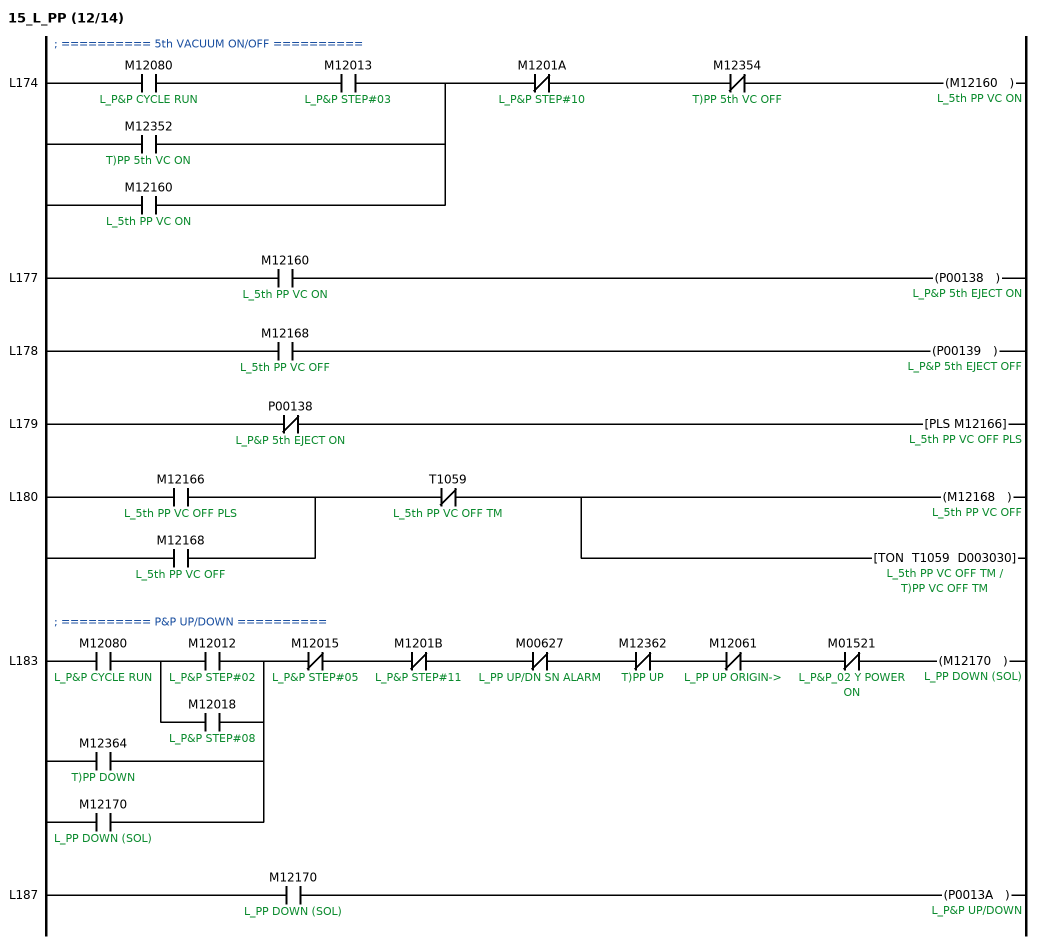
// ========== 5th VACUUM ON/OFF ==========
; L174
LOAD      M12080	// L_P&P CYCLE RUN
AND       M12013	// L_P&P STEP#03
OR        M12352	// T)PP 5th VC ON
OR        M12160	// L_5th PP VC ON
AND NOT   M1201A	// L_P&P STEP#10
AND NOT   M12354	// T)PP 5th VC OFF
OUT       M12160	// L_5th PP VC ON
; L177
LOAD      M12160	// L_5th PP VC ON
OUT       P00138	// L_P&P 5th EJECT ON
; L178
LOAD      M12168	// L_5th PP VC OFF
OUT       P00139	// L_P&P 5th EJECT OFF
; L179
LOAD NOT  P00138	// L_P&P 5th EJECT ON
OUTP      M12166	// L_5th PP VC OFF PLS
; L180
LOAD      M12166	// L_5th PP VC OFF PLS
OR        M12168	// L_5th PP VC OFF
AND NOT   T1059	// L_5th PP VC OFF TM
OUT       M12168	// L_5th PP VC OFF
TON       T1059 D003030	// L_5th PP VC OFF TM / T)PP VC OFF TM
// ========== P&P UP/DOWN ==========
; L183
LOAD      M12080	// L_P&P CYCLE RUN
LOAD      M12012	// L_P&P STEP#02
OR        M12018	// L_P&P STEP#08
AND LOAD
OR        M12364	// T)PP DOWN
OR        M12170	// L_PP DOWN (SOL)
AND NOT   M12015	// L_P&P STEP#05
AND NOT   M1201B	// L_P&P STEP#11
AND NOT   M00627	// L_PP UP/DN SN ALARM
AND NOT   M12362	// T)PP UP
AND NOT   M12061	// L_PP UP ORIGIN->
AND NOT   M01521	// L_P&P_02 Y POWER ON
OUT       M12170	// L_PP DOWN (SOL)
; L187
LOAD      M12170	// L_PP DOWN (SOL)
OUT       P0013A	// L_P&P UP/DOWN

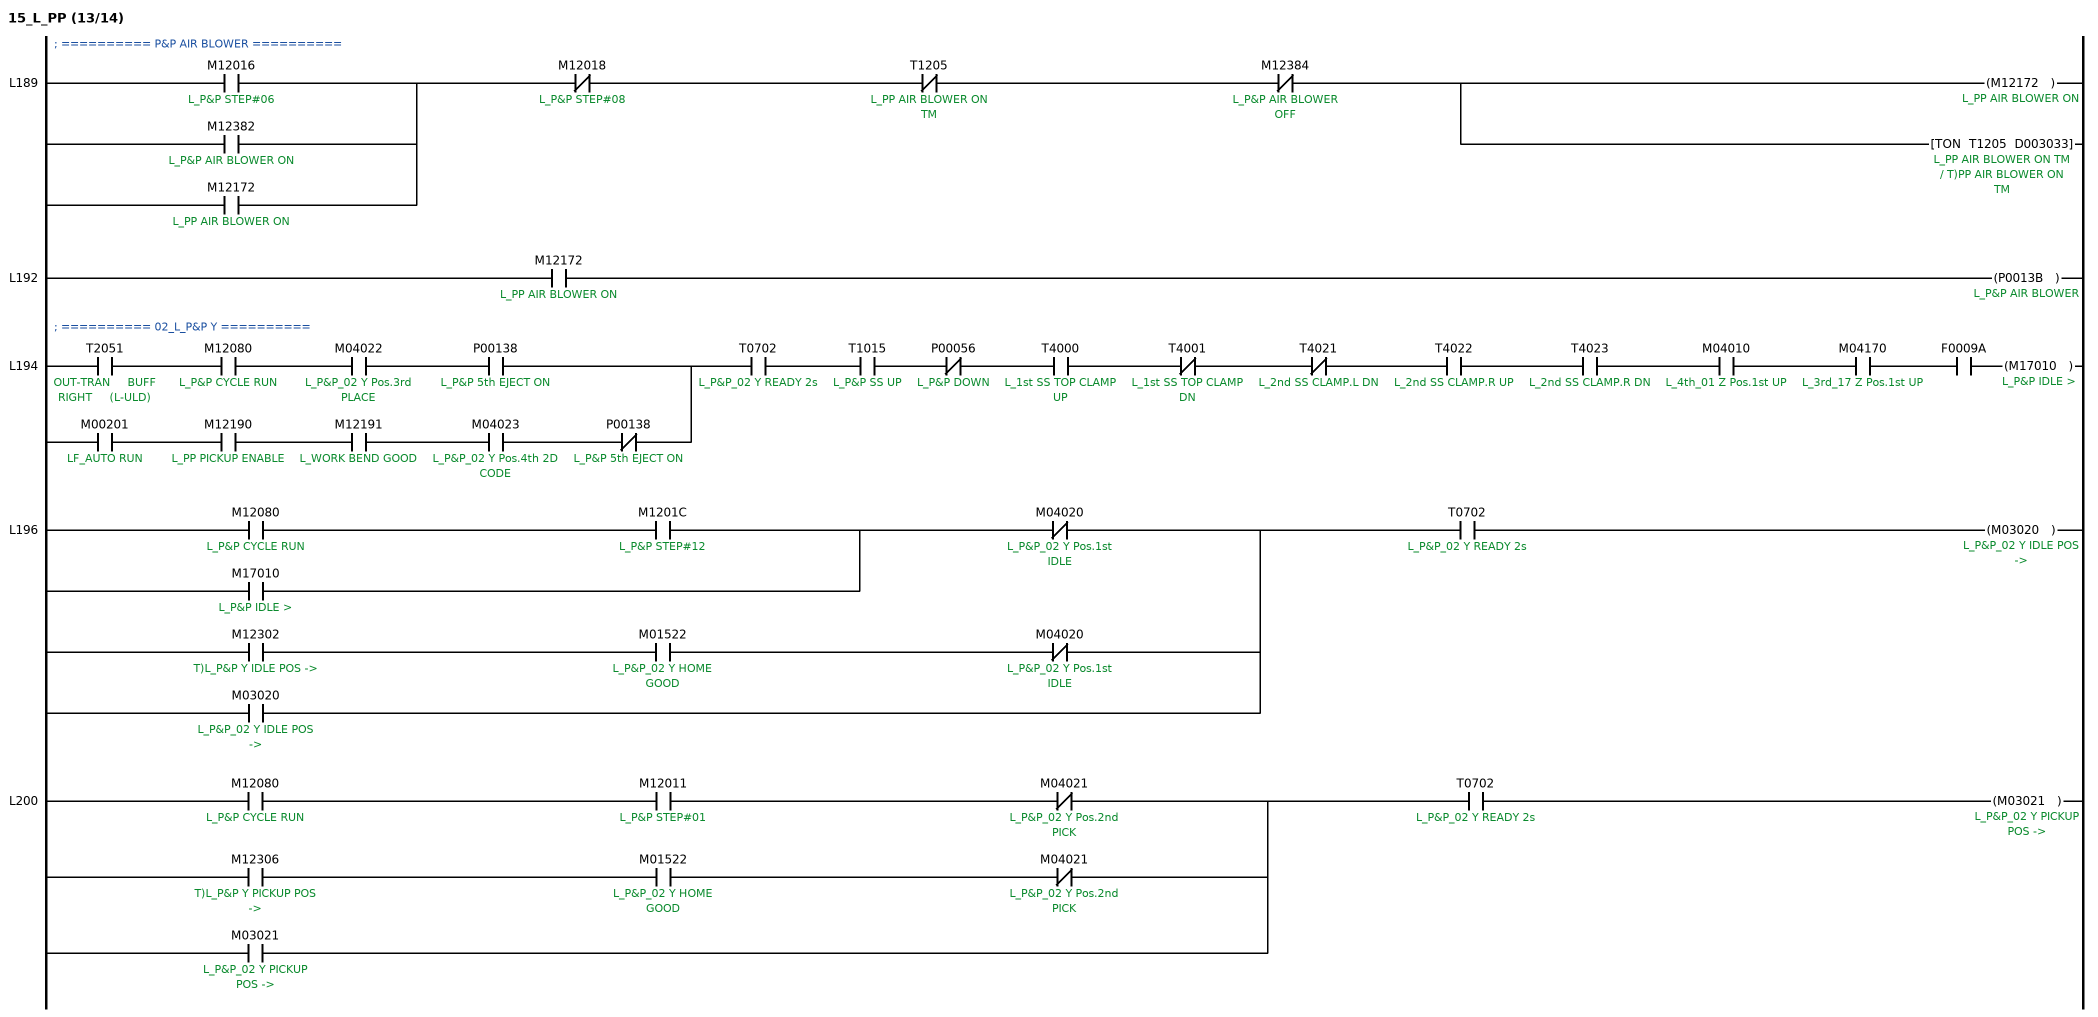
// ========== P&P AIR BLOWER ==========
; L189
LOAD      M12016	// L_P&P STEP#06
OR        M12382	// L_P&P AIR BLOWER ON
OR        M12172	// L_PP AIR BLOWER ON
AND NOT   M12018	// L_P&P STEP#08
AND NOT   T1205	// L_PP AIR BLOWER ON TM
AND NOT   M12384	// L_P&P AIR BLOWER OFF
OUT       M12172	// L_PP AIR BLOWER ON
TON       T1205 D003033	// L_PP AIR BLOWER ON TM / T)PP AIR BLOWER ON TM
; L192
LOAD      M12172	// L_PP AIR BLOWER ON
OUT       P0013B	// L_P&P AIR BLOWER
// ========== 02_L_P&P Y ==========
; L194
LOAD      T2051	// OUT-TRAN     BUFF     RIGHT     (L-ULD)
AND       M12080	// L_P&P CYCLE RUN
AND       M04022	// L_P&P_02 Y Pos.3rd PLACE
AND       P00138	// L_P&P 5th EJECT ON
LOAD      M00201	// LF_AUTO RUN
AND       M12190	// L_PP PICKUP ENABLE
AND       M12191	// L_WORK BEND GOOD
AND       M04023	// L_P&P_02 Y Pos.4th 2D CODE
AND NOT   P00138	// L_P&P 5th EJECT ON
OR LOAD
AND       T0702	// L_P&P_02 Y READY 2s
AND       T1015	// L_P&P SS UP
AND NOT   P00056	// L_P&P DOWN
AND       T4000	// L_1st SS TOP CLAMP    UP
AND NOT   T4001	// L_1st SS TOP CLAMP    DN
AND NOT   T4021	// L_2nd SS CLAMP.L DN
AND       T4022	// L_2nd SS CLAMP.R UP
AND       T4023	// L_2nd SS CLAMP.R DN
AND       M04010	// L_4th_01 Z Pos.1st UP
AND       M04170	// L_3rd_17 Z Pos.1st UP
AND       F0009A
OUT       M17010	// L_P&P IDLE >
; L196
LOAD      M12080	// L_P&P CYCLE RUN
AND       M1201C	// L_P&P STEP#12
OR        M17010	// L_P&P IDLE >
AND NOT   M04020	// L_P&P_02 Y Pos.1st IDLE
LOAD      M12302	// T)L_P&P Y IDLE POS ->
AND       M01522	// L_P&P_02 Y HOME GOOD
AND NOT   M04020	// L_P&P_02 Y Pos.1st IDLE
OR LOAD
OR        M03020	// L_P&P_02 Y IDLE POS ->
AND       T0702	// L_P&P_02 Y READY 2s
OUT       M03020	// L_P&P_02 Y IDLE POS ->
; L200
LOAD      M12080	// L_P&P CYCLE RUN
AND       M12011	// L_P&P STEP#01
AND NOT   M04021	// L_P&P_02 Y Pos.2nd PICK
LOAD      M12306	// T)L_P&P Y PICKUP POS ->
AND       M01522	// L_P&P_02 Y HOME GOOD
AND NOT   M04021	// L_P&P_02 Y Pos.2nd PICK
OR LOAD
OR        M03021	// L_P&P_02 Y PICKUP POS ->
AND       T0702	// L_P&P_02 Y READY 2s
OUT       M03021	// L_P&P_02 Y PICKUP POS ->

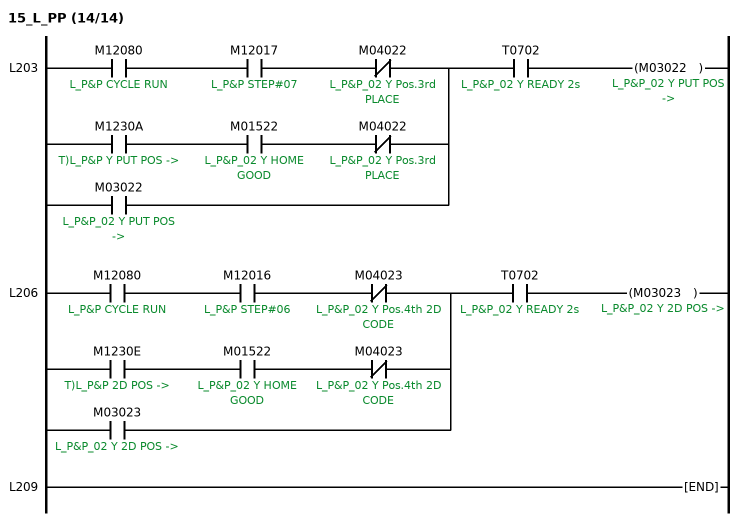
; L203
LOAD      M12080	// L_P&P CYCLE RUN
AND       M12017	// L_P&P STEP#07
AND NOT   M04022	// L_P&P_02 Y Pos.3rd PLACE
LOAD      M1230A	// T)L_P&P Y PUT POS ->
AND       M01522	// L_P&P_02 Y HOME GOOD
AND NOT   M04022	// L_P&P_02 Y Pos.3rd PLACE
OR LOAD
OR        M03022	// L_P&P_02 Y PUT POS ->
AND       T0702	// L_P&P_02 Y READY 2s
OUT       M03022	// L_P&P_02 Y PUT POS ->
; L206
LOAD      M12080	// L_P&P CYCLE RUN
AND       M12016	// L_P&P STEP#06
AND NOT   M04023	// L_P&P_02 Y Pos.4th 2D CODE
LOAD      M1230E	// T)L_P&P 2D POS ->
AND       M01522	// L_P&P_02 Y HOME GOOD
AND NOT   M04023	// L_P&P_02 Y Pos.4th 2D CODE
OR LOAD
OR        M03023	// L_P&P_02 Y 2D POS ->
AND       T0702	// L_P&P_02 Y READY 2s
OUT       M03023	// L_P&P_02 Y 2D POS ->
; L209
END

PROGRAM 16_R_1st_MAND (task: ¨ö¨¬A¥ì CA¡¤I¡¾¡¿¡¤¡Í)

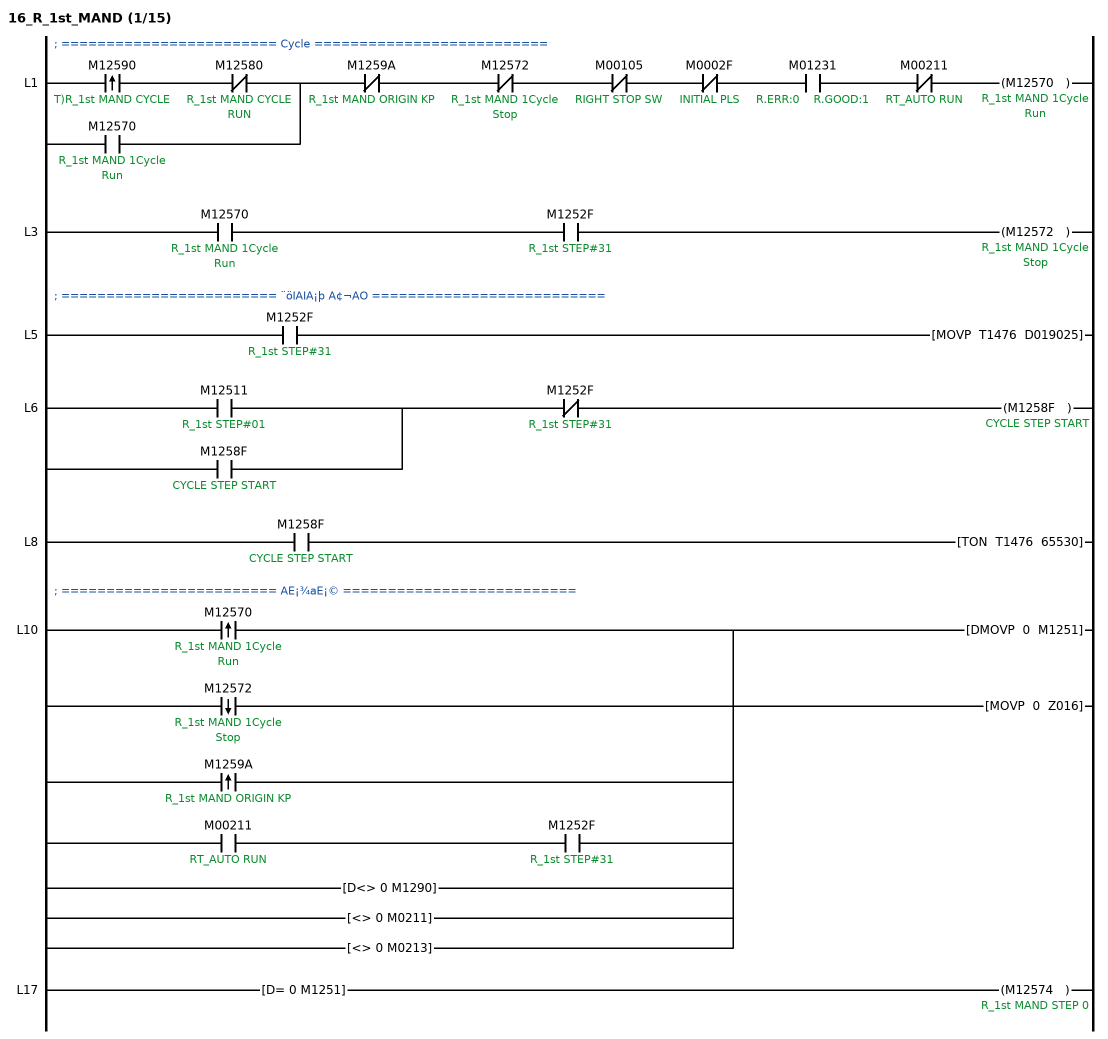
// ======================== Cycle ==========================
; L1
LOADP     M12590	// T)R_1st MAND CYCLE
AND NOT   M12580	// R_1st MAND CYCLE RUN
OR        M12570	// R_1st MAND 1Cycle Run
AND NOT   M1259A	// R_1st MAND ORIGIN KP
AND NOT   M12572	// R_1st MAND 1Cycle Stop
AND NOT   M00105	// RIGHT STOP SW
AND NOT   M0002F	// INITIAL PLS
AND       M01231	// R.ERR:0    R.GOOD:1
AND NOT   M00211	// RT_AUTO RUN
OUT       M12570	// R_1st MAND 1Cycle Run
; L3
LOAD      M12570	// R_1st MAND 1Cycle Run
AND       M1252F	// R_1st STEP#31
OUT       M12572	// R_1st MAND 1Cycle Stop
// ======================== ¨öIAIA¡þ A¢¬AO ==========================
; L5
LOAD      M1252F	// R_1st STEP#31
MOVP      T1476 D019025
; L6
LOAD      M12511	// R_1st STEP#01
OR        M1258F	// CYCLE STEP START
AND NOT   M1252F	// R_1st STEP#31
OUT       M1258F	// CYCLE STEP START
; L8
LOAD      M1258F	// CYCLE STEP START
TON       T1476 65530
// ======================== AE¡¾aE¡© ==========================
; L10
LOADP     M12570	// R_1st MAND 1Cycle Run
ORN       M12572	// R_1st MAND 1Cycle Stop
ORP       M1259A	// R_1st MAND ORIGIN KP
LOAD      M00211	// RT_AUTO RUN
AND       M1252F	// R_1st STEP#31
OR LOAD
ORD<>     0 M1290
OR<>      0 M0211
OR<>      0 M0213
DMOVP     0 M1251
MOVP      0 Z016
; L17
LOADD=    0 M1251
OUT       M12574	// R_1st MAND STEP 0

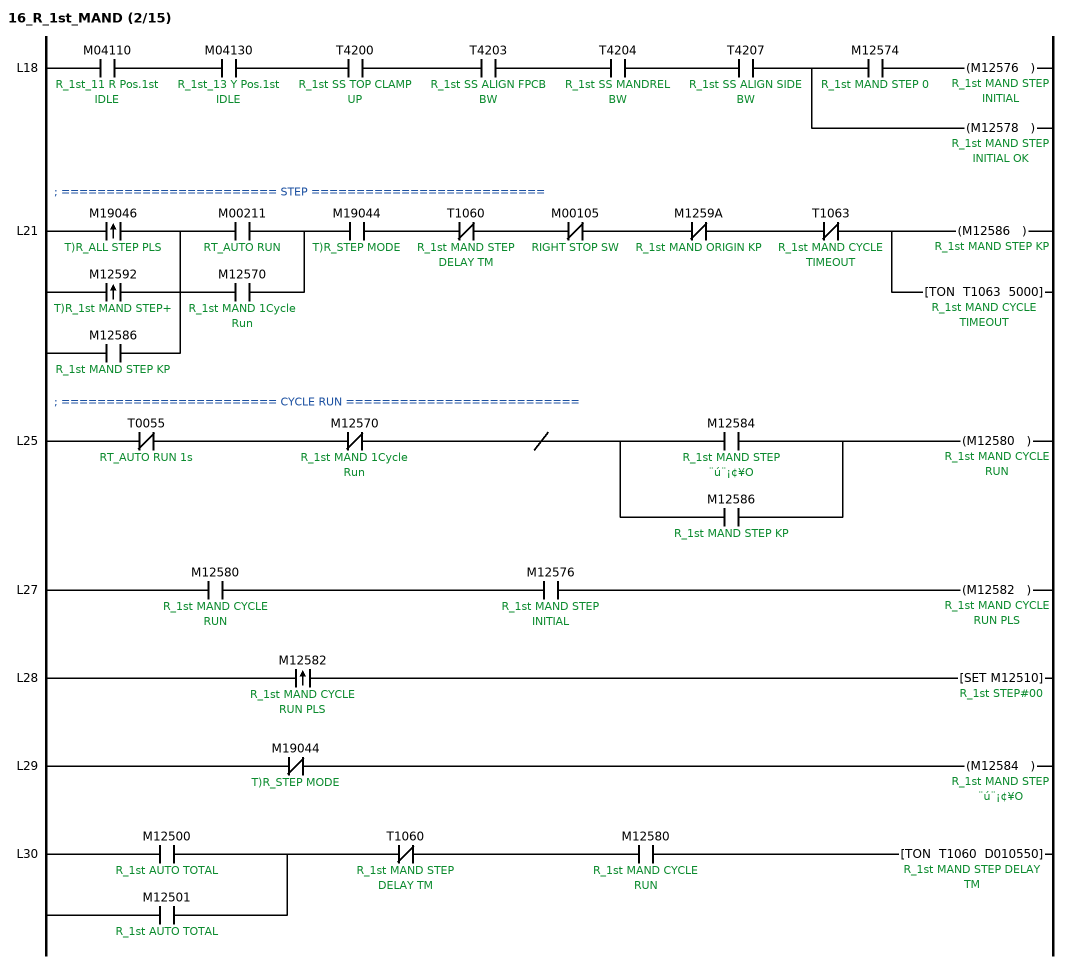
; L18
LOAD      M04110	// R_1st_11 R Pos.1st IDLE
AND       M04130	// R_1st_13 Y Pos.1st IDLE
AND       T4200	// R_1st SS TOP CLAMP UP
AND       T4203	// R_1st SS ALIGN FPCB BW
AND       T4204	// R_1st SS MANDREL BW
AND       T4207	// R_1st SS ALIGN SIDE BW
MPUSH
AND       M12574	// R_1st MAND STEP 0
OUT       M12576	// R_1st MAND STEP INITIAL
MPOP
OUT       M12578	// R_1st MAND STEP INITIAL OK
// ======================== STEP ==========================
; L21
LOADP     M19046	// T)R_ALL STEP PLS
ORP       M12592	// T)R_1st MAND STEP+
OR        M12586	// R_1st MAND STEP KP
LOAD      M00211	// RT_AUTO RUN
OR        M12570	// R_1st MAND 1Cycle Run
AND LOAD
AND       M19044	// T)R_STEP MODE
AND NOT   T1060	// R_1st MAND STEP DELAY TM
AND NOT   M00105	// RIGHT STOP SW
AND NOT   M1259A	// R_1st MAND ORIGIN KP
AND NOT   T1063	// R_1st MAND CYCLE TIMEOUT
OUT       M12586	// R_1st MAND STEP KP
TON       T1063 5000	// R_1st MAND CYCLE TIMEOUT
// ======================== CYCLE RUN ==========================
; L25
LOAD NOT  T0055	// RT_AUTO RUN 1s
AND NOT   M12570	// R_1st MAND 1Cycle Run
NOT
LOAD      M12584	// R_1st MAND STEP ¨ú¨¡¢¥O
OR        M12586	// R_1st MAND STEP KP
AND LOAD
OUT       M12580	// R_1st MAND CYCLE RUN
; L27
LOAD      M12580	// R_1st MAND CYCLE RUN
AND       M12576	// R_1st MAND STEP INITIAL
OUT       M12582	// R_1st MAND CYCLE RUN PLS
; L28
LOADP     M12582	// R_1st MAND CYCLE RUN PLS
SET       M12510	// R_1st STEP#00
; L29
LOAD NOT  M19044	// T)R_STEP MODE
OUT       M12584	// R_1st MAND STEP ¨ú¨¡¢¥O
; L30
LOAD      M12500	// R_1st AUTO TOTAL
OR        M12501	// R_1st AUTO TOTAL
AND NOT   T1060	// R_1st MAND STEP DELAY TM
AND       M12580	// R_1st MAND CYCLE RUN
TON       T1060 D010550	// R_1st MAND STEP DELAY TM

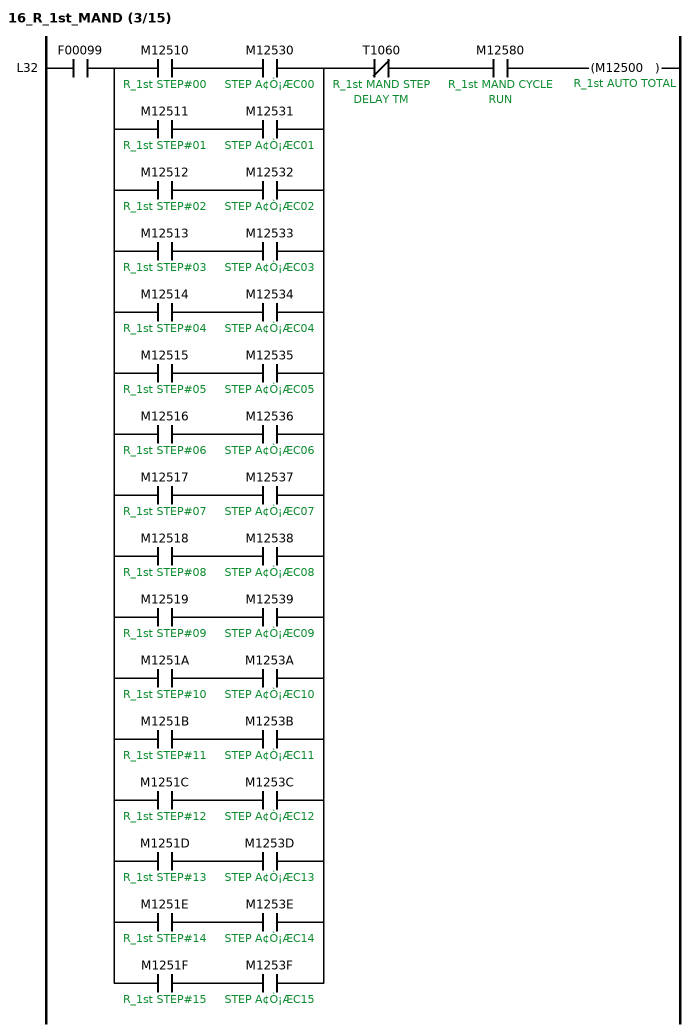
; L32
LOAD      F00099
LOAD      M12510	// R_1st STEP#00
AND       M12530	// STEP A¢Ò¡ÆC00
LOAD      M12511	// R_1st STEP#01
AND       M12531	// STEP A¢Ò¡ÆC01
OR LOAD
LOAD      M12512	// R_1st STEP#02
AND       M12532	// STEP A¢Ò¡ÆC02
OR LOAD
LOAD      M12513	// R_1st STEP#03
AND       M12533	// STEP A¢Ò¡ÆC03
OR LOAD
LOAD      M12514	// R_1st STEP#04
AND       M12534	// STEP A¢Ò¡ÆC04
OR LOAD
LOAD      M12515	// R_1st STEP#05
AND       M12535	// STEP A¢Ò¡ÆC05
OR LOAD
LOAD      M12516	// R_1st STEP#06
AND       M12536	// STEP A¢Ò¡ÆC06
OR LOAD
LOAD      M12517	// R_1st STEP#07
AND       M12537	// STEP A¢Ò¡ÆC07
OR LOAD
LOAD      M12518	// R_1st STEP#08
AND       M12538	// STEP A¢Ò¡ÆC08
OR LOAD
LOAD      M12519	// R_1st STEP#09
AND       M12539	// STEP A¢Ò¡ÆC09
OR LOAD
LOAD      M1251A	// R_1st STEP#10
AND       M1253A	// STEP A¢Ò¡ÆC10
OR LOAD
LOAD      M1251B	// R_1st STEP#11
AND       M1253B	// STEP A¢Ò¡ÆC11
OR LOAD
LOAD      M1251C	// R_1st STEP#12
AND       M1253C	// STEP A¢Ò¡ÆC12
OR LOAD
LOAD      M1251D	// R_1st STEP#13
AND       M1253D	// STEP A¢Ò¡ÆC13
OR LOAD
LOAD      M1251E	// R_1st STEP#14
AND       M1253E	// STEP A¢Ò¡ÆC14
OR LOAD
LOAD      M1251F	// R_1st STEP#15
AND       M1253F	// STEP A¢Ò¡ÆC15
OR LOAD
AND LOAD
AND NOT   T1060	// R_1st MAND STEP DELAY TM
AND       M12580	// R_1st MAND CYCLE RUN
OUT       M12500	// R_1st AUTO TOTAL

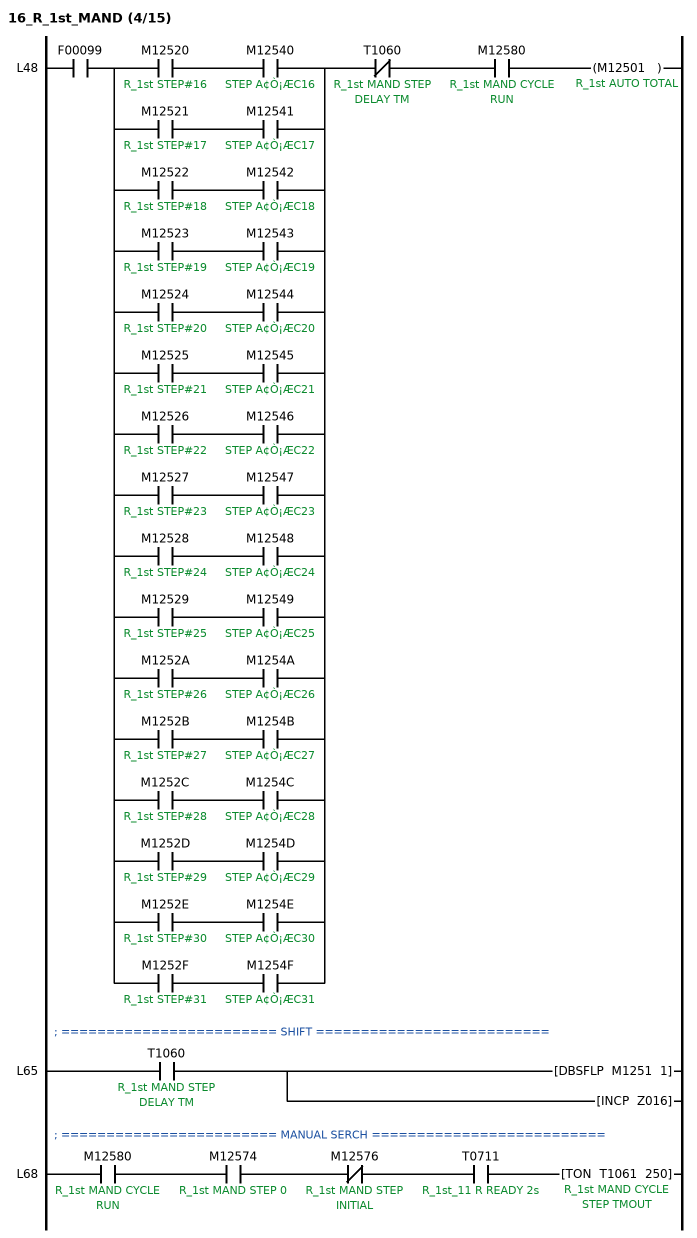
; L48
LOAD      F00099
LOAD      M12520	// R_1st STEP#16
AND       M12540	// STEP A¢Ò¡ÆC16
LOAD      M12521	// R_1st STEP#17
AND       M12541	// STEP A¢Ò¡ÆC17
OR LOAD
LOAD      M12522	// R_1st STEP#18
AND       M12542	// STEP A¢Ò¡ÆC18
OR LOAD
LOAD      M12523	// R_1st STEP#19
AND       M12543	// STEP A¢Ò¡ÆC19
OR LOAD
LOAD      M12524	// R_1st STEP#20
AND       M12544	// STEP A¢Ò¡ÆC20
OR LOAD
LOAD      M12525	// R_1st STEP#21
AND       M12545	// STEP A¢Ò¡ÆC21
OR LOAD
LOAD      M12526	// R_1st STEP#22
AND       M12546	// STEP A¢Ò¡ÆC22
OR LOAD
LOAD      M12527	// R_1st STEP#23
AND       M12547	// STEP A¢Ò¡ÆC23
OR LOAD
LOAD      M12528	// R_1st STEP#24
AND       M12548	// STEP A¢Ò¡ÆC24
OR LOAD
LOAD      M12529	// R_1st STEP#25
AND       M12549	// STEP A¢Ò¡ÆC25
OR LOAD
LOAD      M1252A	// R_1st STEP#26
AND       M1254A	// STEP A¢Ò¡ÆC26
OR LOAD
LOAD      M1252B	// R_1st STEP#27
AND       M1254B	// STEP A¢Ò¡ÆC27
OR LOAD
LOAD      M1252C	// R_1st STEP#28
AND       M1254C	// STEP A¢Ò¡ÆC28
OR LOAD
LOAD      M1252D	// R_1st STEP#29
AND       M1254D	// STEP A¢Ò¡ÆC29
OR LOAD
LOAD      M1252E	// R_1st STEP#30
AND       M1254E	// STEP A¢Ò¡ÆC30
OR LOAD
LOAD      M1252F	// R_1st STEP#31
AND       M1254F	// STEP A¢Ò¡ÆC31
OR LOAD
AND LOAD
AND NOT   T1060	// R_1st MAND STEP DELAY TM
AND       M12580	// R_1st MAND CYCLE RUN
OUT       M12501	// R_1st AUTO TOTAL
// ======================== SHIFT ==========================
; L65
LOAD      T1060	// R_1st MAND STEP DELAY TM
DBSFLP    M1251 1
INCP      Z016
// ======================== MANUAL SERCH ==========================
; L68
LOAD      M12580	// R_1st MAND CYCLE RUN
AND       M12574	// R_1st MAND STEP 0
AND NOT   M12576	// R_1st MAND STEP INITIAL
AND       T0711	// R_1st_11 R READY 2s
TON       T1061 250	// R_1st MAND CYCLE STEP TMOUT

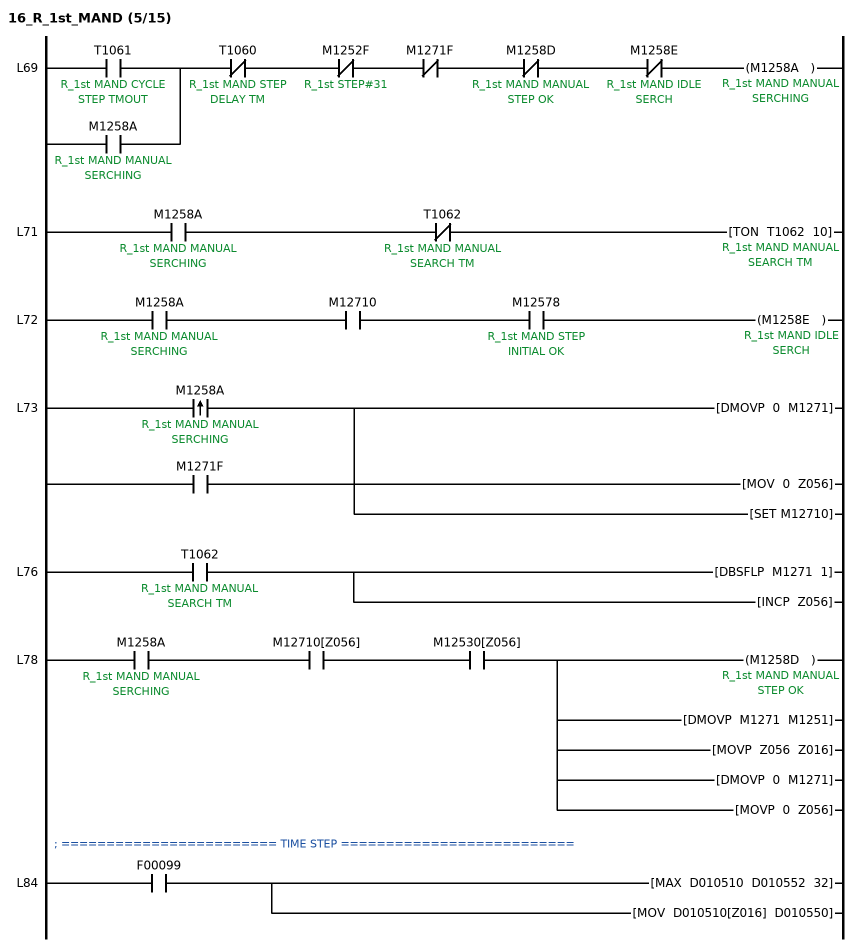
; L69
LOAD      T1061	// R_1st MAND CYCLE STEP TMOUT
OR        M1258A	// R_1st MAND MANUAL SERCHING
AND NOT   T1060	// R_1st MAND STEP DELAY TM
AND NOT   M1252F	// R_1st STEP#31
AND NOT   M1271F
AND NOT   M1258D	// R_1st MAND MANUAL STEP OK
AND NOT   M1258E	// R_1st MAND IDLE SERCH
OUT       M1258A	// R_1st MAND MANUAL SERCHING
; L71
LOAD      M1258A	// R_1st MAND MANUAL SERCHING
AND NOT   T1062	// R_1st MAND MANUAL SEARCH TM
TON       T1062 10	// R_1st MAND MANUAL SEARCH TM
; L72
LOAD      M1258A	// R_1st MAND MANUAL SERCHING
AND       M12710
AND       M12578	// R_1st MAND STEP INITIAL OK
OUT       M1258E	// R_1st MAND IDLE SERCH
; L73
LOADP     M1258A	// R_1st MAND MANUAL SERCHING
OR        M1271F
DMOVP     0 M1271
MOV       0 Z056
SET       M12710
; L76
LOAD      T1062	// R_1st MAND MANUAL SEARCH TM
DBSFLP    M1271 1
INCP      Z056
; L78
LOAD      M1258A	// R_1st MAND MANUAL SERCHING
AND       M12710[Z056]
AND       M12530[Z056]
OUT       M1258D	// R_1st MAND MANUAL STEP OK
DMOVP     M1271 M1251
MOVP      Z056 Z016
DMOVP     0 M1271
MOVP      0 Z056
// ======================== TIME STEP ==========================
; L84
LOAD      F00099
MAX       D010510 D010552 32
MOV       D010510[Z016] D010550

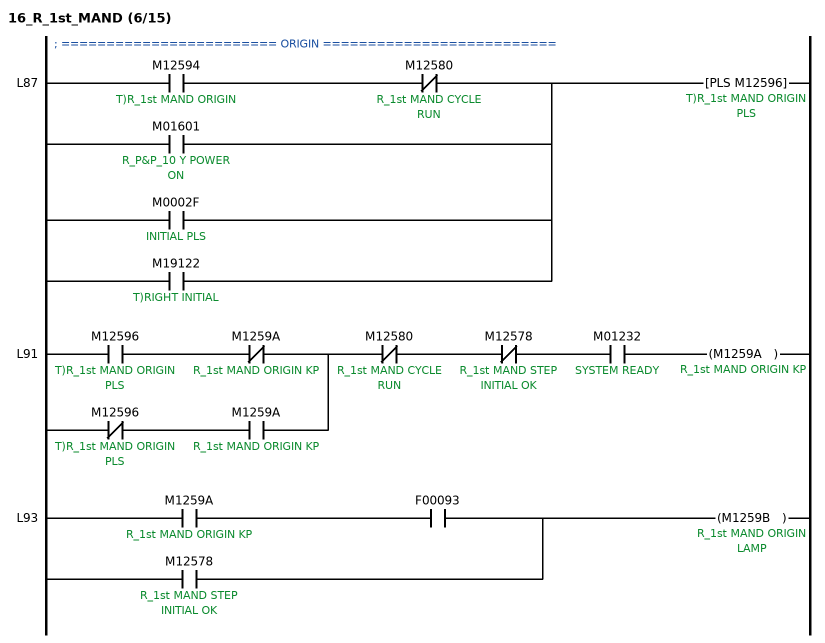
// ======================== ORIGIN ==========================
; L87
LOAD      M12594	// T)R_1st MAND ORIGIN
AND NOT   M12580	// R_1st MAND CYCLE RUN
OR        M01601	// R_P&P_10 Y POWER ON
OR        M0002F	// INITIAL PLS
OR        M19122	// T)RIGHT INITIAL
OUTP      M12596	// T)R_1st MAND ORIGIN PLS
; L91
LOAD      M12596	// T)R_1st MAND ORIGIN PLS
AND NOT   M1259A	// R_1st MAND ORIGIN KP
LOAD NOT  M12596	// T)R_1st MAND ORIGIN PLS
AND       M1259A	// R_1st MAND ORIGIN KP
OR LOAD
AND NOT   M12580	// R_1st MAND CYCLE RUN
AND NOT   M12578	// R_1st MAND STEP INITIAL OK
AND       M01232	// SYSTEM READY
OUT       M1259A	// R_1st MAND ORIGIN KP
; L93
LOAD      M1259A	// R_1st MAND ORIGIN KP
AND       F00093
OR        M12578	// R_1st MAND STEP INITIAL OK
OUT       M1259B	// R_1st MAND ORIGIN LAMP

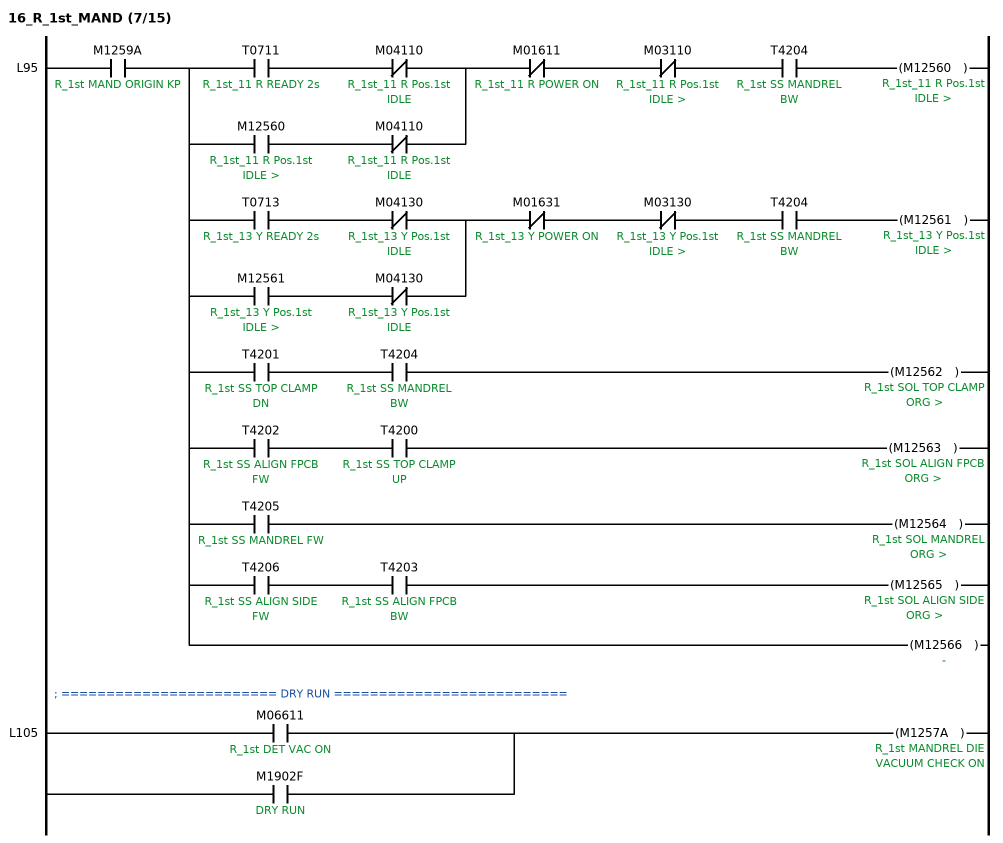
; L95
LOAD      M1259A	// R_1st MAND ORIGIN KP
MPUSH
LOAD      T0711	// R_1st_11 R READY 2s
AND NOT   M04110	// R_1st_11 R Pos.1st IDLE
LOAD      M12560	// R_1st_11 R Pos.1st IDLE >
AND NOT   M04110	// R_1st_11 R Pos.1st IDLE
OR LOAD
AND LOAD
AND NOT   M01611	// R_1st_11 R POWER ON
AND NOT   M03110	// R_1st_11 R Pos.1st IDLE >
AND       T4204	// R_1st SS MANDREL BW
OUT       M12560	// R_1st_11 R Pos.1st IDLE >
MLOAD
LOAD      T0713	// R_1st_13 Y READY 2s
AND NOT   M04130	// R_1st_13 Y Pos.1st IDLE
LOAD      M12561	// R_1st_13 Y Pos.1st IDLE >
AND NOT   M04130	// R_1st_13 Y Pos.1st IDLE
OR LOAD
AND LOAD
AND NOT   M01631	// R_1st_13 Y POWER ON
AND NOT   M03130	// R_1st_13 Y Pos.1st IDLE >
AND       T4204	// R_1st SS MANDREL BW
OUT       M12561	// R_1st_13 Y Pos.1st IDLE >
MLOAD
AND       T4201	// R_1st SS TOP CLAMP DN
AND       T4204	// R_1st SS MANDREL BW
OUT       M12562	// R_1st SOL TOP CLAMP ORG >
MLOAD
AND       T4202	// R_1st SS ALIGN FPCB FW
AND       T4200	// R_1st SS TOP CLAMP UP
OUT       M12563	// R_1st SOL ALIGN FPCB ORG >
MLOAD
AND       T4205	// R_1st SS MANDREL FW
OUT       M12564	// R_1st SOL MANDREL ORG >
MLOAD
AND       T4206	// R_1st SS ALIGN SIDE FW
AND       T4203	// R_1st SS ALIGN FPCB BW
OUT       M12565	// R_1st SOL ALIGN SIDE ORG >
MPOP
OUT       M12566	// -
// ======================== DRY RUN ==========================
; L105
LOAD      M06611	// R_1st DET VAC ON
OR        M1902F	// DRY RUN
OUT       M1257A	// R_1st MANDREL DIE VACUUM CHECK ON

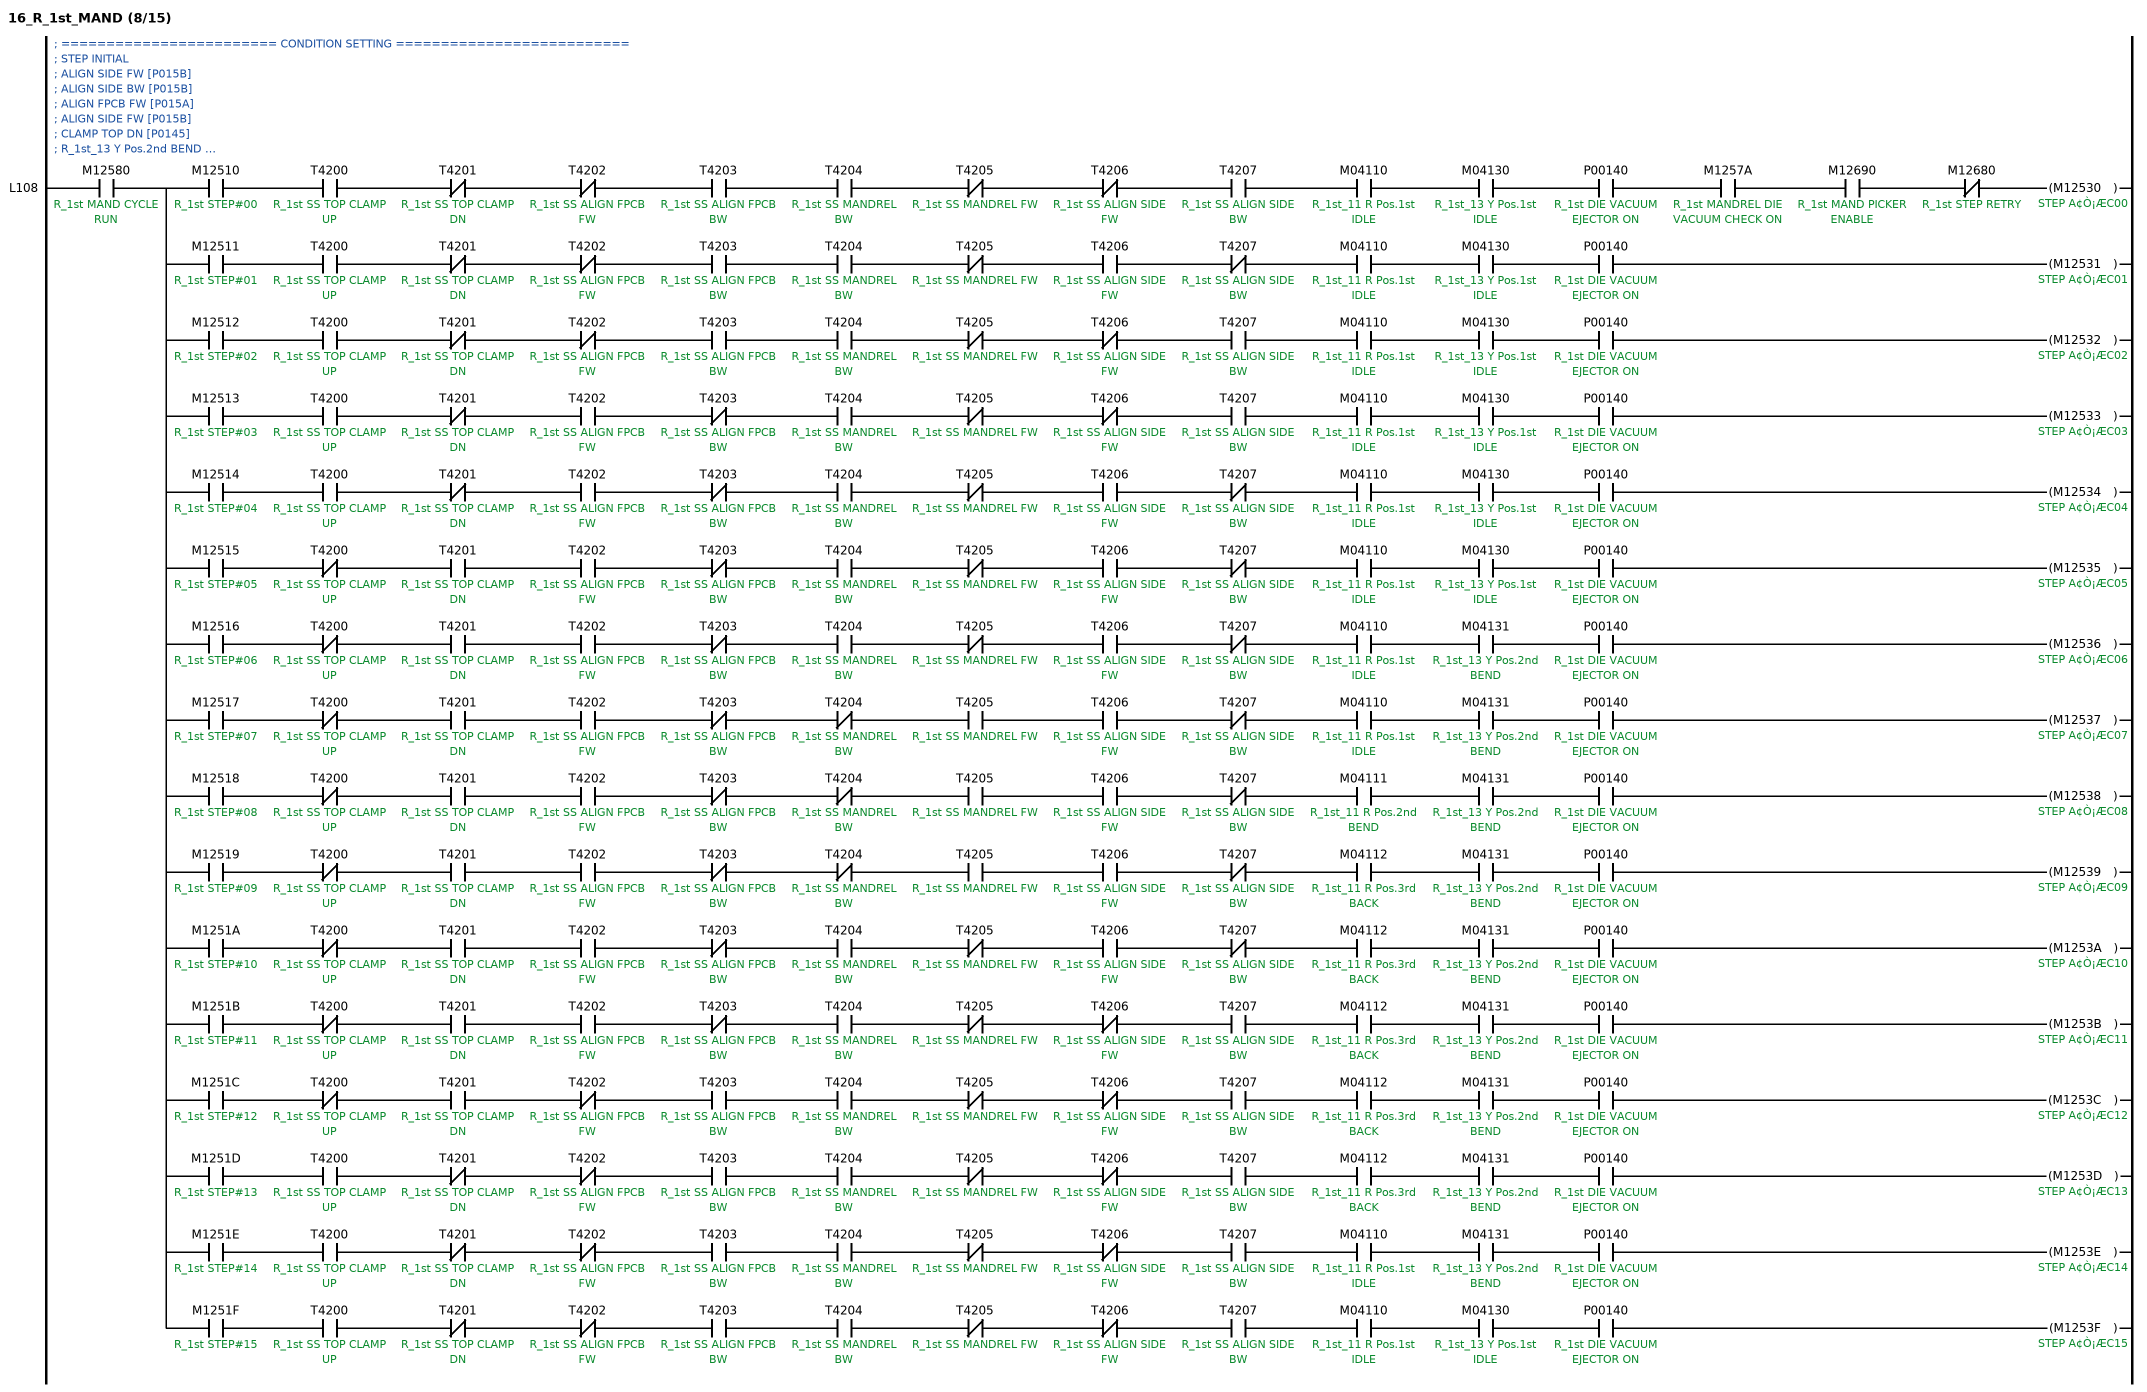
// ======================== CONDITION SETTING ==========================
; L108
LOAD      M12580	// R_1st MAND CYCLE RUN
MPUSH
AND       M12510	// R_1st STEP#00
AND       T4200	// R_1st SS TOP CLAMP UP
AND NOT   T4201	// R_1st SS TOP CLAMP DN
AND NOT   T4202	// R_1st SS ALIGN FPCB FW
AND       T4203	// R_1st SS ALIGN FPCB BW
AND       T4204	// R_1st SS MANDREL BW
AND NOT   T4205	// R_1st SS MANDREL FW
AND NOT   T4206	// R_1st SS ALIGN SIDE FW
AND       T4207	// R_1st SS ALIGN SIDE BW
AND       M04110	// R_1st_11 R Pos.1st IDLE
AND       M04130	// R_1st_13 Y Pos.1st IDLE
AND       P00140	// R_1st DIE VACUUM EJECTOR ON
AND       M1257A	// R_1st MANDREL DIE VACUUM CHECK ON
AND       M12690	// R_1st MAND PICKER ENABLE
AND NOT   M12680	// R_1st STEP RETRY
OUT       M12530	// STEP A¢Ò¡ÆC00
MLOAD
AND       M12511	// R_1st STEP#01
AND       T4200	// R_1st SS TOP CLAMP UP
AND NOT   T4201	// R_1st SS TOP CLAMP DN
AND NOT   T4202	// R_1st SS ALIGN FPCB FW
AND       T4203	// R_1st SS ALIGN FPCB BW
AND       T4204	// R_1st SS MANDREL BW
AND NOT   T4205	// R_1st SS MANDREL FW
AND       T4206	// R_1st SS ALIGN SIDE FW
AND NOT   T4207	// R_1st SS ALIGN SIDE BW
AND       M04110	// R_1st_11 R Pos.1st IDLE
AND       M04130	// R_1st_13 Y Pos.1st IDLE
AND       P00140	// R_1st DIE VACUUM EJECTOR ON
OUT       M12531	// STEP A¢Ò¡ÆC01
MLOAD
AND       M12512	// R_1st STEP#02
AND       T4200	// R_1st SS TOP CLAMP UP
AND NOT   T4201	// R_1st SS TOP CLAMP DN
AND NOT   T4202	// R_1st SS ALIGN FPCB FW
AND       T4203	// R_1st SS ALIGN FPCB BW
AND       T4204	// R_1st SS MANDREL BW
AND NOT   T4205	// R_1st SS MANDREL FW
AND NOT   T4206	// R_1st SS ALIGN SIDE FW
AND       T4207	// R_1st SS ALIGN SIDE BW
AND       M04110	// R_1st_11 R Pos.1st IDLE
AND       M04130	// R_1st_13 Y Pos.1st IDLE
AND       P00140	// R_1st DIE VACUUM EJECTOR ON
OUT       M12532	// STEP A¢Ò¡ÆC02
MLOAD
AND       M12513	// R_1st STEP#03
AND       T4200	// R_1st SS TOP CLAMP UP
AND NOT   T4201	// R_1st SS TOP CLAMP DN
AND       T4202	// R_1st SS ALIGN FPCB FW
AND NOT   T4203	// R_1st SS ALIGN FPCB BW
AND       T4204	// R_1st SS MANDREL BW
AND NOT   T4205	// R_1st SS MANDREL FW
AND NOT   T4206	// R_1st SS ALIGN SIDE FW
AND       T4207	// R_1st SS ALIGN SIDE BW
AND       M04110	// R_1st_11 R Pos.1st IDLE
AND       M04130	// R_1st_13 Y Pos.1st IDLE
AND       P00140	// R_1st DIE VACUUM EJECTOR ON
OUT       M12533	// STEP A¢Ò¡ÆC03
MLOAD
AND       M12514	// R_1st STEP#04
AND       T4200	// R_1st SS TOP CLAMP UP
AND NOT   T4201	// R_1st SS TOP CLAMP DN
AND       T4202	// R_1st SS ALIGN FPCB FW
AND NOT   T4203	// R_1st SS ALIGN FPCB BW
AND       T4204	// R_1st SS MANDREL BW
AND NOT   T4205	// R_1st SS MANDREL FW
AND       T4206	// R_1st SS ALIGN SIDE FW
AND NOT   T4207	// R_1st SS ALIGN SIDE BW
AND       M04110	// R_1st_11 R Pos.1st IDLE
AND       M04130	// R_1st_13 Y Pos.1st IDLE
AND       P00140	// R_1st DIE VACUUM EJECTOR ON
OUT       M12534	// STEP A¢Ò¡ÆC04
MLOAD
AND       M12515	// R_1st STEP#05
AND NOT   T4200	// R_1st SS TOP CLAMP UP
AND       T4201	// R_1st SS TOP CLAMP DN
AND       T4202	// R_1st SS ALIGN FPCB FW
AND NOT   T4203	// R_1st SS ALIGN FPCB BW
AND       T4204	// R_1st SS MANDREL BW
AND NOT   T4205	// R_1st SS MANDREL FW
AND       T4206	// R_1st SS ALIGN SIDE FW
AND NOT   T4207	// R_1st SS ALIGN SIDE BW
AND       M04110	// R_1st_11 R Pos.1st IDLE
AND       M04130	// R_1st_13 Y Pos.1st IDLE
AND       P00140	// R_1st DIE VACUUM EJECTOR ON
OUT       M12535	// STEP A¢Ò¡ÆC05
MLOAD
AND       M12516	// R_1st STEP#06
AND NOT   T4200	// R_1st SS TOP CLAMP UP
AND       T4201	// R_1st SS TOP CLAMP DN
AND       T4202	// R_1st SS ALIGN FPCB FW
AND NOT   T4203	// R_1st SS ALIGN FPCB BW
AND       T4204	// R_1st SS MANDREL BW
AND NOT   T4205	// R_1st SS MANDREL FW
AND       T4206	// R_1st SS ALIGN SIDE FW
AND NOT   T4207	// R_1st SS ALIGN SIDE BW
AND       M04110	// R_1st_11 R Pos.1st IDLE
AND       M04131	// R_1st_13 Y Pos.2nd BEND
AND       P00140	// R_1st DIE VACUUM EJECTOR ON
OUT       M12536	// STEP A¢Ò¡ÆC06
MLOAD
AND       M12517	// R_1st STEP#07
AND NOT   T4200	// R_1st SS TOP CLAMP UP
AND       T4201	// R_1st SS TOP CLAMP DN
AND       T4202	// R_1st SS ALIGN FPCB FW
AND NOT   T4203	// R_1st SS ALIGN FPCB BW
AND NOT   T4204	// R_1st SS MANDREL BW
AND       T4205	// R_1st SS MANDREL FW
AND       T4206	// R_1st SS ALIGN SIDE FW
AND NOT   T4207	// R_1st SS ALIGN SIDE BW
AND       M04110	// R_1st_11 R Pos.1st IDLE
AND       M04131	// R_1st_13 Y Pos.2nd BEND
AND       P00140	// R_1st DIE VACUUM EJECTOR ON
OUT       M12537	// STEP A¢Ò¡ÆC07
MLOAD
AND       M12518	// R_1st STEP#08
AND NOT   T4200	// R_1st SS TOP CLAMP UP
AND       T4201	// R_1st SS TOP CLAMP DN
AND       T4202	// R_1st SS ALIGN FPCB FW
AND NOT   T4203	// R_1st SS ALIGN FPCB BW
AND NOT   T4204	// R_1st SS MANDREL BW
AND       T4205	// R_1st SS MANDREL FW
AND       T4206	// R_1st SS ALIGN SIDE FW
AND NOT   T4207	// R_1st SS ALIGN SIDE BW
AND       M04111	// R_1st_11 R Pos.2nd BEND
AND       M04131	// R_1st_13 Y Pos.2nd BEND
AND       P00140	// R_1st DIE VACUUM EJECTOR ON
OUT       M12538	// STEP A¢Ò¡ÆC08
MLOAD
AND       M12519	// R_1st STEP#09
AND NOT   T4200	// R_1st SS TOP CLAMP UP
AND       T4201	// R_1st SS TOP CLAMP DN
AND       T4202	// R_1st SS ALIGN FPCB FW
AND NOT   T4203	// R_1st SS ALIGN FPCB BW
AND NOT   T4204	// R_1st SS MANDREL BW
AND       T4205	// R_1st SS MANDREL FW
AND       T4206	// R_1st SS ALIGN SIDE FW
AND NOT   T4207	// R_1st SS ALIGN SIDE BW
AND       M04112	// R_1st_11 R Pos.3rd BACK
AND       M04131	// R_1st_13 Y Pos.2nd BEND
AND       P00140	// R_1st DIE VACUUM EJECTOR ON
OUT       M12539	// STEP A¢Ò¡ÆC09
MLOAD
AND       M1251A	// R_1st STEP#10
AND NOT   T4200	// R_1st SS TOP CLAMP UP
AND       T4201	// R_1st SS TOP CLAMP DN
AND       T4202	// R_1st SS ALIGN FPCB FW
AND NOT   T4203	// R_1st SS ALIGN FPCB BW
AND       T4204	// R_1st SS MANDREL BW
AND NOT   T4205	// R_1st SS MANDREL FW
AND       T4206	// R_1st SS ALIGN SIDE FW
AND NOT   T4207	// R_1st SS ALIGN SIDE BW
AND       M04112	// R_1st_11 R Pos.3rd BACK
AND       M04131	// R_1st_13 Y Pos.2nd BEND
AND       P00140	// R_1st DIE VACUUM EJECTOR ON
OUT       M1253A	// STEP A¢Ò¡ÆC10
MLOAD
AND       M1251B	// R_1st STEP#11
AND NOT   T4200	// R_1st SS TOP CLAMP UP
AND       T4201	// R_1st SS TOP CLAMP DN
AND       T4202	// R_1st SS ALIGN FPCB FW
AND NOT   T4203	// R_1st SS ALIGN FPCB BW
AND       T4204	// R_1st SS MANDREL BW
AND NOT   T4205	// R_1st SS MANDREL FW
AND NOT   T4206	// R_1st SS ALIGN SIDE FW
AND       T4207	// R_1st SS ALIGN SIDE BW
AND       M04112	// R_1st_11 R Pos.3rd BACK
AND       M04131	// R_1st_13 Y Pos.2nd BEND
AND       P00140	// R_1st DIE VACUUM EJECTOR ON
OUT       M1253B	// STEP A¢Ò¡ÆC11
MLOAD
AND       M1251C	// R_1st STEP#12
AND NOT   T4200	// R_1st SS TOP CLAMP UP
AND       T4201	// R_1st SS TOP CLAMP DN
AND NOT   T4202	// R_1st SS ALIGN FPCB FW
AND       T4203	// R_1st SS ALIGN FPCB BW
AND       T4204	// R_1st SS MANDREL BW
AND NOT   T4205	// R_1st SS MANDREL FW
AND NOT   T4206	// R_1st SS ALIGN SIDE FW
AND       T4207	// R_1st SS ALIGN SIDE BW
AND       M04112	// R_1st_11 R Pos.3rd BACK
AND       M04131	// R_1st_13 Y Pos.2nd BEND
AND       P00140	// R_1st DIE VACUUM EJECTOR ON
OUT       M1253C	// STEP A¢Ò¡ÆC12
MLOAD
AND       M1251D	// R_1st STEP#13
AND       T4200	// R_1st SS TOP CLAMP UP
AND NOT   T4201	// R_1st SS TOP CLAMP DN
AND NOT   T4202	// R_1st SS ALIGN FPCB FW
AND       T4203	// R_1st SS ALIGN FPCB BW
AND       T4204	// R_1st SS MANDREL BW
AND NOT   T4205	// R_1st SS MANDREL FW
AND NOT   T4206	// R_1st SS ALIGN SIDE FW
AND       T4207	// R_1st SS ALIGN SIDE BW
AND       M04112	// R_1st_11 R Pos.3rd BACK
AND       M04131	// R_1st_13 Y Pos.2nd BEND
AND       P00140	// R_1st DIE VACUUM EJECTOR ON
OUT       M1253D	// STEP A¢Ò¡ÆC13
MLOAD
AND       M1251E	// R_1st STEP#14
AND       T4200	// R_1st SS TOP CLAMP UP
AND NOT   T4201	// R_1st SS TOP CLAMP DN
AND NOT   T4202	// R_1st SS ALIGN FPCB FW
AND       T4203	// R_1st SS ALIGN FPCB BW
AND       T4204	// R_1st SS MANDREL BW
AND NOT   T4205	// R_1st SS MANDREL FW
AND NOT   T4206	// R_1st SS ALIGN SIDE FW
AND       T4207	// R_1st SS ALIGN SIDE BW
AND       M04110	// R_1st_11 R Pos.1st IDLE
AND       M04131	// R_1st_13 Y Pos.2nd BEND
AND       P00140	// R_1st DIE VACUUM EJECTOR ON
OUT       M1253E	// STEP A¢Ò¡ÆC14
MPOP
AND       M1251F	// R_1st STEP#15
AND       T4200	// R_1st SS TOP CLAMP UP
AND NOT   T4201	// R_1st SS TOP CLAMP DN
AND NOT   T4202	// R_1st SS ALIGN FPCB FW
AND       T4203	// R_1st SS ALIGN FPCB BW
AND       T4204	// R_1st SS MANDREL BW
AND NOT   T4205	// R_1st SS MANDREL FW
AND NOT   T4206	// R_1st SS ALIGN SIDE FW
AND       T4207	// R_1st SS ALIGN SIDE BW
AND       M04110	// R_1st_11 R Pos.1st IDLE
AND       M04130	// R_1st_13 Y Pos.1st IDLE
AND       P00140	// R_1st DIE VACUUM EJECTOR ON
OUT       M1253F	// STEP A¢Ò¡ÆC15
// output comment: STEP INITIAL
// output comment: ALIGN SIDE FW [P015B]
// output comment: ALIGN SIDE BW [P015B]
// output comment: ALIGN FPCB FW [P015A]
// output comment: ALIGN SIDE FW [P015B]
// output comment: CLAMP TOP DN [P0145]
// output comment: R_1st_13 Y Pos.2nd BEND >
// output comment: MANDREL FW        [P0144]
// output comment: R_1st_11 R Pos.2nd BEND >
// output comment: R_1st_11 R Pos.3rd BACK >
// output comment: MANDREL BW     [P0144]
// output comment: ALIGN SIDE BW [P015B]
// output comment: ALIGN FPCB BW [P015A]
// output comment: CLAMP TOP UP [P0145]
// output comment: R_1st_11 R Pos.1st IDLE >
// output comment: R_1st_13 Y Pos.1st IDLE >

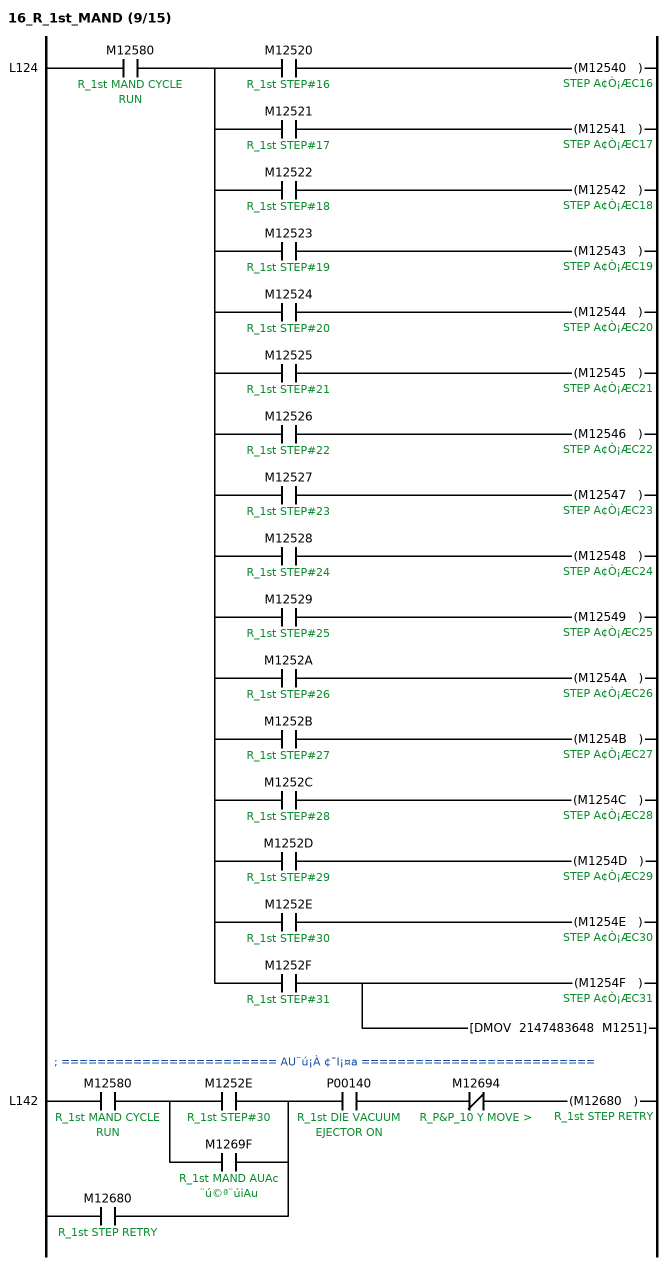
; L124
LOAD      M12580	// R_1st MAND CYCLE RUN
MPUSH
AND       M12520	// R_1st STEP#16
OUT       M12540	// STEP A¢Ò¡ÆC16
MLOAD
AND       M12521	// R_1st STEP#17
OUT       M12541	// STEP A¢Ò¡ÆC17
MLOAD
AND       M12522	// R_1st STEP#18
OUT       M12542	// STEP A¢Ò¡ÆC18
MLOAD
AND       M12523	// R_1st STEP#19
OUT       M12543	// STEP A¢Ò¡ÆC19
MLOAD
AND       M12524	// R_1st STEP#20
OUT       M12544	// STEP A¢Ò¡ÆC20
MLOAD
AND       M12525	// R_1st STEP#21
OUT       M12545	// STEP A¢Ò¡ÆC21
MLOAD
AND       M12526	// R_1st STEP#22
OUT       M12546	// STEP A¢Ò¡ÆC22
MLOAD
AND       M12527	// R_1st STEP#23
OUT       M12547	// STEP A¢Ò¡ÆC23
MLOAD
AND       M12528	// R_1st STEP#24
OUT       M12548	// STEP A¢Ò¡ÆC24
MLOAD
AND       M12529	// R_1st STEP#25
OUT       M12549	// STEP A¢Ò¡ÆC25
MLOAD
AND       M1252A	// R_1st STEP#26
OUT       M1254A	// STEP A¢Ò¡ÆC26
MLOAD
AND       M1252B	// R_1st STEP#27
OUT       M1254B	// STEP A¢Ò¡ÆC27
MLOAD
AND       M1252C	// R_1st STEP#28
OUT       M1254C	// STEP A¢Ò¡ÆC28
MLOAD
AND       M1252D	// R_1st STEP#29
OUT       M1254D	// STEP A¢Ò¡ÆC29
MLOAD
AND       M1252E	// R_1st STEP#30
OUT       M1254E	// STEP A¢Ò¡ÆC30
MPOP
AND       M1252F	// R_1st STEP#31
OUT       M1254F	// STEP A¢Ò¡ÆC31
DMOV      2147483648 M1251
// ======================== AU¨ú¡À ¢¯I¡¤a ==========================
; L142
LOAD      M12580	// R_1st MAND CYCLE RUN
LOAD      M1252E	// R_1st STEP#30
OR        M1269F	// R_1st MAND AUAc ¨ú©ª¨úiAu
AND LOAD
OR        M12680	// R_1st STEP RETRY
AND       P00140	// R_1st DIE VACUUM EJECTOR ON
AND NOT   M12694	// R_P&P_10 Y MOVE >
OUT       M12680	// R_1st STEP RETRY

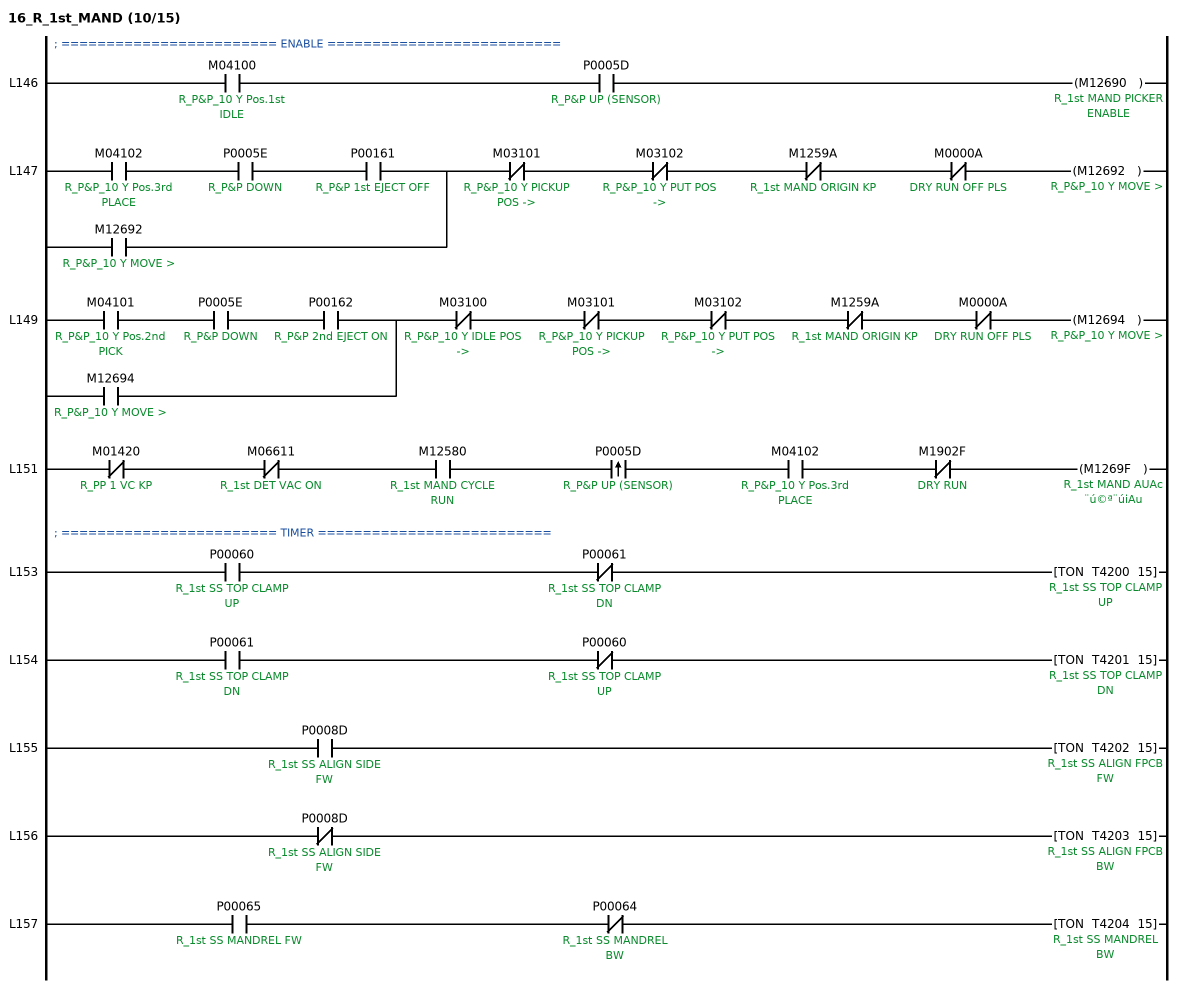
// ======================== ENABLE ==========================
; L146
LOAD      M04100	// R_P&P_10 Y Pos.1st IDLE
AND       P0005D	// R_P&P UP (SENSOR)
OUT       M12690	// R_1st MAND PICKER ENABLE
; L147
LOAD      M04102	// R_P&P_10 Y Pos.3rd PLACE
AND       P0005E	// R_P&P DOWN
AND       P00161	// R_P&P 1st EJECT OFF
OR        M12692	// R_P&P_10 Y MOVE >
AND NOT   M03101	// R_P&P_10 Y PICKUP POS ->
AND NOT   M03102	// R_P&P_10 Y PUT POS ->
AND NOT   M1259A	// R_1st MAND ORIGIN KP
AND NOT   M0000A	// DRY RUN OFF PLS
OUT       M12692	// R_P&P_10 Y MOVE >
; L149
LOAD      M04101	// R_P&P_10 Y Pos.2nd PICK
AND       P0005E	// R_P&P DOWN
AND       P00162	// R_P&P 2nd EJECT ON
OR        M12694	// R_P&P_10 Y MOVE >
AND NOT   M03100	// R_P&P_10 Y IDLE POS ->
AND NOT   M03101	// R_P&P_10 Y PICKUP POS ->
AND NOT   M03102	// R_P&P_10 Y PUT POS ->
AND NOT   M1259A	// R_1st MAND ORIGIN KP
AND NOT   M0000A	// DRY RUN OFF PLS
OUT       M12694	// R_P&P_10 Y MOVE >
; L151
LOAD NOT  M01420	// R_PP 1 VC KP
AND NOT   M06611	// R_1st DET VAC ON
AND       M12580	// R_1st MAND CYCLE RUN
ANDP      P0005D	// R_P&P UP (SENSOR)
AND       M04102	// R_P&P_10 Y Pos.3rd PLACE
AND NOT   M1902F	// DRY RUN
OUT       M1269F	// R_1st MAND AUAc ¨ú©ª¨úiAu
// ======================== TIMER ==========================
; L153
LOAD      P00060	// R_1st SS TOP CLAMP UP
AND NOT   P00061	// R_1st SS TOP CLAMP DN
TON       T4200 15	// R_1st SS TOP CLAMP UP
; L154
LOAD      P00061	// R_1st SS TOP CLAMP DN
AND NOT   P00060	// R_1st SS TOP CLAMP UP
TON       T4201 15	// R_1st SS TOP CLAMP DN
; L155
LOAD      P0008D	// R_1st SS ALIGN SIDE FW
TON       T4202 15	// R_1st SS ALIGN FPCB FW
; L156
LOAD NOT  P0008D	// R_1st SS ALIGN SIDE FW
TON       T4203 15	// R_1st SS ALIGN FPCB BW
; L157
LOAD      P00065	// R_1st SS MANDREL FW
AND NOT   P00064	// R_1st SS MANDREL BW
TON       T4204 15	// R_1st SS MANDREL BW

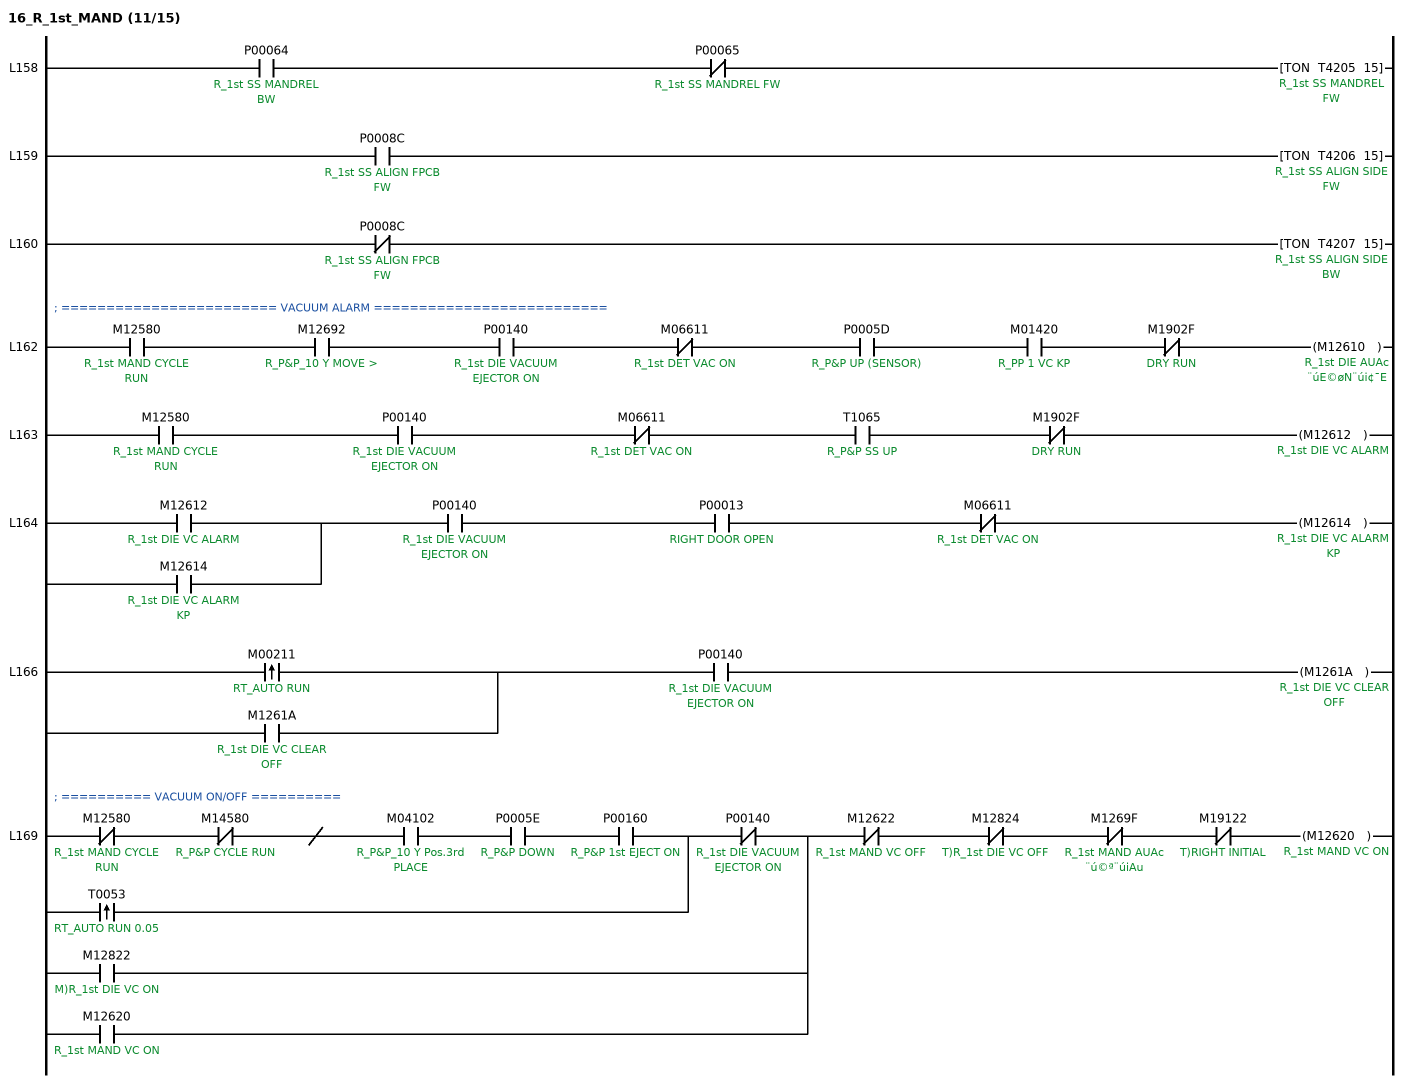
; L158
LOAD      P00064	// R_1st SS MANDREL BW
AND NOT   P00065	// R_1st SS MANDREL FW
TON       T4205 15	// R_1st SS MANDREL FW
; L159
LOAD      P0008C	// R_1st SS ALIGN FPCB FW
TON       T4206 15	// R_1st SS ALIGN SIDE FW
; L160
LOAD NOT  P0008C	// R_1st SS ALIGN FPCB FW
TON       T4207 15	// R_1st SS ALIGN SIDE BW
// ======================== VACUUM ALARM ==========================
; L162
LOAD      M12580	// R_1st MAND CYCLE RUN
AND       M12692	// R_P&P_10 Y MOVE >
AND       P00140	// R_1st DIE VACUUM EJECTOR ON
AND NOT   M06611	// R_1st DET VAC ON
AND       P0005D	// R_P&P UP (SENSOR)
AND       M01420	// R_PP 1 VC KP
AND NOT   M1902F	// DRY RUN
OUT       M12610	// R_1st DIE AUAc ¨úE©øN¨úi¢¯E
; L163
LOAD      M12580	// R_1st MAND CYCLE RUN
AND       P00140	// R_1st DIE VACUUM EJECTOR ON
AND NOT   M06611	// R_1st DET VAC ON
AND       T1065	// R_P&P SS UP
AND NOT   M1902F	// DRY RUN
OUT       M12612	// R_1st DIE VC ALARM
; L164
LOAD      M12612	// R_1st DIE VC ALARM
OR        M12614	// R_1st DIE VC ALARM KP
AND       P00140	// R_1st DIE VACUUM EJECTOR ON
AND       P00013	// RIGHT DOOR OPEN
AND NOT   M06611	// R_1st DET VAC ON
OUT       M12614	// R_1st DIE VC ALARM KP
; L166
LOADP     M00211	// RT_AUTO RUN
OR        M1261A	// R_1st DIE VC CLEAR OFF
AND       P00140	// R_1st DIE VACUUM EJECTOR ON
OUT       M1261A	// R_1st DIE VC CLEAR OFF
// ========== VACUUM ON/OFF ==========
; L169
LOAD NOT  M12580	// R_1st MAND CYCLE RUN
AND NOT   M14580	// R_P&P CYCLE RUN
NOT
AND       M04102	// R_P&P_10 Y Pos.3rd PLACE
AND       P0005E	// R_P&P DOWN
AND       P00160	// R_P&P 1st EJECT ON
ORP       T0053	// RT_AUTO RUN 0.05
AND NOT   P00140	// R_1st DIE VACUUM EJECTOR ON
OR        M12822	// M)R_1st DIE VC ON
OR        M12620	// R_1st MAND VC ON
AND NOT   M12622	// R_1st MAND VC OFF
AND NOT   M12824	// T)R_1st DIE VC OFF
AND NOT   M1269F	// R_1st MAND AUAc ¨ú©ª¨úiAu
AND NOT   M19122	// T)RIGHT INITIAL
OUT       M12620	// R_1st MAND VC ON

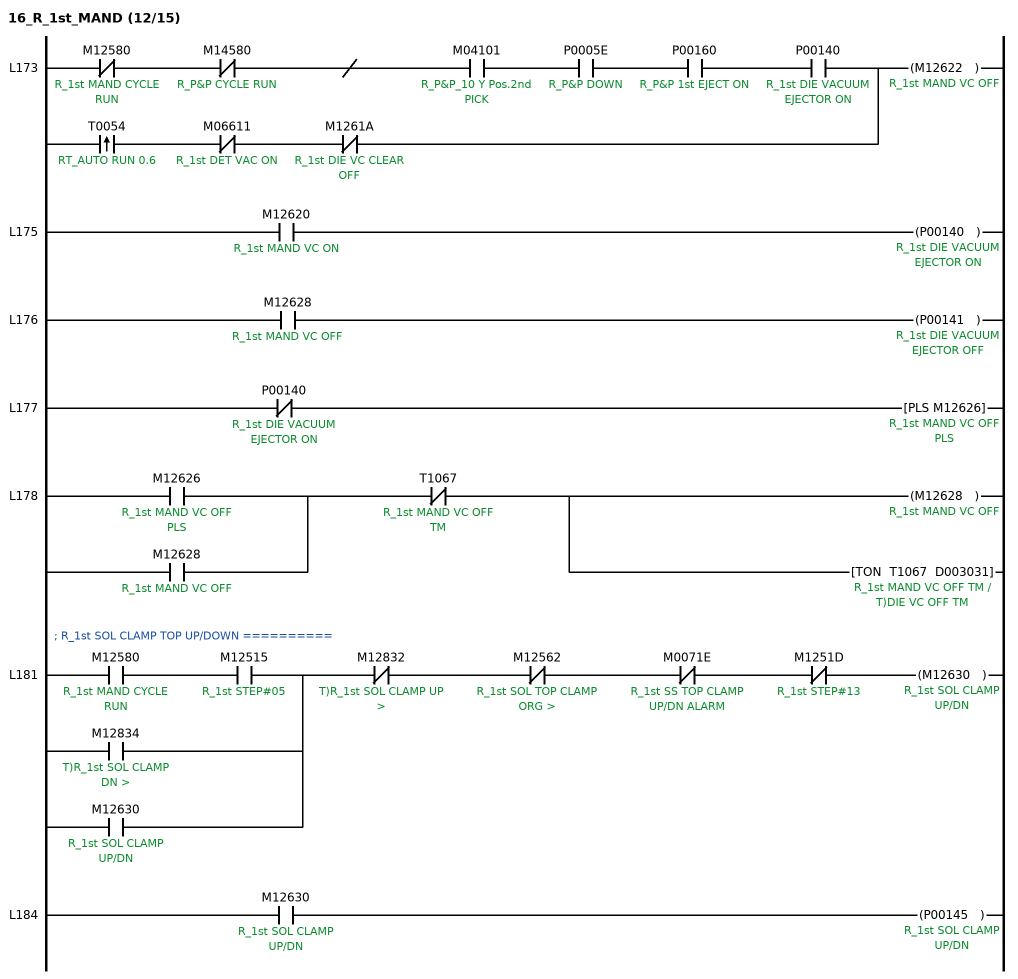
; L173
LOAD NOT  M12580	// R_1st MAND CYCLE RUN
AND NOT   M14580	// R_P&P CYCLE RUN
NOT
AND       M04101	// R_P&P_10 Y Pos.2nd PICK
AND       P0005E	// R_P&P DOWN
AND       P00160	// R_P&P 1st EJECT ON
AND       P00140	// R_1st DIE VACUUM EJECTOR ON
LOADP     T0054	// RT_AUTO RUN 0.6
AND NOT   M06611	// R_1st DET VAC ON
AND NOT   M1261A	// R_1st DIE VC CLEAR OFF
OR LOAD
OUT       M12622	// R_1st MAND VC OFF
; L175
LOAD      M12620	// R_1st MAND VC ON
OUT       P00140	// R_1st DIE VACUUM EJECTOR ON
; L176
LOAD      M12628	// R_1st MAND VC OFF
OUT       P00141	// R_1st DIE VACUUM EJECTOR OFF
; L177
LOAD NOT  P00140	// R_1st DIE VACUUM EJECTOR ON
OUTP      M12626	// R_1st MAND VC OFF PLS
; L178
LOAD      M12626	// R_1st MAND VC OFF PLS
OR        M12628	// R_1st MAND VC OFF
AND NOT   T1067	// R_1st MAND VC OFF TM
OUT       M12628	// R_1st MAND VC OFF
TON       T1067 D003031	// R_1st MAND VC OFF TM / T)DIE VC OFF TM
//  R_1st SOL CLAMP TOP UP/DOWN ==========
; L181
LOAD      M12580	// R_1st MAND CYCLE RUN
AND       M12515	// R_1st STEP#05
OR        M12834	// T)R_1st SOL CLAMP DN >
OR        M12630	// R_1st SOL CLAMP UP/DN
AND NOT   M12832	// T)R_1st SOL CLAMP UP >
AND NOT   M12562	// R_1st SOL TOP CLAMP ORG >
AND NOT   M0071E	// R_1st SS TOP CLAMP UP/DN ALARM
AND NOT   M1251D	// R_1st STEP#13
OUT       M12630	// R_1st SOL CLAMP UP/DN
; L184
LOAD      M12630	// R_1st SOL CLAMP UP/DN
OUT       P00145	// R_1st SOL CLAMP UP/DN

